LIN {X 0,Y 359.947,Z 582.419,A -85,B 0,C 180,E1 -13482.824,E2 -13482.824} C_VEL
LIN {X 0,Y 358.594,Z 592.161,A -85,B 0,C 180,E1 -13484.075,E2 -13484.075} C_VEL
LIN {X 0,Y 357.358,Z 601.086,A -85,B 0,C 180,E1 -13485.478,E2 -13485.478} C_VEL
LIN {X 0,Y 356.154,Z 609.872,A -85,B 0,C 180,E1 -13487.174,E2 -13487.174} C_VEL
LIN {X 0,Y 355.202,Z 616.932,A -85,B 0,C 180,E1 -13488.877,E2 -13488.877} C_VEL
LIN {X 0,Y 354.322,Z 623.413,A -85,B 0,C 180,E1 -13490.87,E2 -13490.87} C_VEL
LIN {X 0,Y 353.781,Z 627.649,A -85,B 0,C 180,E1 -13492.581,E2 -13492.581} C_VEL
LIN {X 0,Y 353.502,Z 630.768,A -85,B 0,C 180,E1 -13494.295,E2 -13494.295} C_VEL
LIN {X 0,Y 353.381,Z 632.27,A -85,B 0,C 180,E1 -13495.437,E2 -13495.437} C_VEL
LIN {X 0,Y 353.229,Z 633.321,A -85,B 0,C 180,E1 -13496.578,E2 -13496.578} C_VEL
LIN {X 0,Y 353.155,Z 633.956,A -85,B 0,C 180,E1 -13497.719,E2 -13497.719} C_VEL
LIN {X 0,Y 353.153,Z 634.14,A -85,B 0,C 180,E1 -13498.86,E2 -13498.86} C_VEL
LIN {X 0,Y 353.146,Z 633.86,A -85,B 0,C 180,E1 -13500,E2 -13500} C_VEL
LIN {X 0,Y 353.151,Z 633.161,A -85,B 0,C 180,E1 -13501.14,E2 -13501.14} C_VEL
LIN {X 0,Y 353.141,Z 632.017,A -85,B 0,C 180,E1 -13502.281,E2 -13502.281} C_VEL
LIN {X 0,Y 353.281,Z 629.42,A -85,B 0,C 180,E1 -13503.993,E2 -13503.993} C_VEL
LIN {X 0,Y 353.393,Z 624.752,A -85,B 0,C 180,E1 -13506.079,E2 -13506.079} C_VEL
LIN {X 0,Y 353.647,Z 618.898,A -85,B 0,C 180,E1 -13507.996,E2 -13507.996} C_VEL
LIN {X 0,Y 354.026,Z 612.126,A -85,B 0,C 180,E1 -13509.715,E2 -13509.715} C_VEL
LIN {X 0,Y 354.548,Z 603.69,A -85,B 0,C 180,E1 -13511.433,E2 -13511.433} C_VEL
LIN {X 0,Y 355.239,Z 595.006,A -85,B 0,C 180,E1 -13512.86,E2 -13512.86} C_VEL
LIN {X 0,Y 356,Z 584.552,A -85,B 0,C 180,E1 -13514.264,E2 -13514.264} C_VEL
LIN {X 0,Y 356.698,Z 573.904,A -85,B 0,C 180,E1 -13515.425,E2 -13515.425} C_VEL
LIN {X 0,Y 357.436,Z 562.446,A -85,B 0,C 180,E1 -13516.418,E2 -13516.418} C_VEL
LIN {X 0,Y 358.135,Z 549.906,A -85,B 0,C 180,E1 -13517.266,E2 -13517.266} C_VEL
LIN {X 0,Y 358.795,Z 536.113,A -85,B 0,C 180,E1 -13517.933,E2 -13517.933} C_VEL
LIN {X 0,Y 359.155,Z 522.822,A -85,B 0,C 180,E1 -13518.356,E2 -13518.356} C_VEL
LIN {X 0,Y 361.016,Z 446.902,A -85,B 0,C 180,E1 -13520.357,E2 -13520.357} C_VEL
LIN {X 0,Y 357.928,Z 420.522,A -85,B 0,C 180,E1 -13521.225,E2 -13521.225} C_VEL
LIN {X 0,Y 359.275,Z 398.729,A -85,B 0,C 180,E1 -13524.871,E2 -13524.871} C_VEL
LIN {X 0,Y 360.508,Z 380.834,A -85,B 0,C 180,E1 -13527.897,E2 -13527.897} C_VEL
LIN {X 0,Y 358.657,Z 371.766,A -85,B 0,C 180,E1 -13529.579,E2 -13529.579} C_VEL
LIN {X 0,Y 354.853,Z 355.064,A -85,B 0,C 180,E1 -13532.79,E2 -13532.79} C_VEL
LIN {X 0,Y 354.803,Z 354.916,A -85,B 0,C 180,E1 -13536.459,E2 -13536.459} C_VEL
LIN {X 0,Y 354.83,Z 354.91,A -85,B 0,C 180,E1 -13539.423,E2 -13539.423} C_VEL
LIN {X 0,Y 354.794,Z 354.909,A -85,B 0,C 180,E1 -13542.867,E2 -13542.867} C_VEL
LIN {X 0,Y 354.772,Z 354.901,A -85,B 0,C 180,E1 -13546.103,E2 -13546.103} C_VEL
LIN {X 0,Y 354.793,Z 354.906,A -85,B 0,C 180,E1 -13549.178,E2 -13549.178} C_VEL
LIN {X 0,Y 354.818,Z 354.914,A -85,B 0,C 180,E1 -13552.401,E2 -13552.401} C_VEL
LIN {X 0,Y 354.818,Z 354.904,A -85,B 0,C 180,E1 -13554.94,E2 -13554.94} C_VEL
LIN {X 0,Y 354.862,Z 355.109,A -85,B 0,C 180,E1 -13557.978,E2 -13557.978} C_VEL
LIN {X 0,Y 357.702,Z 366.862,A -85,B 0,C 180,E1 -13561.224,E2 -13561.224} C_VEL
LIN {X 0,Y 358.904,Z 372.282,A -85,B 0,C 180,E1 -13562.587,E2 -13562.587} C_VEL
LIN {X 0,Y 364.389,Z 385.82,A -85,B 0,C 180,E1 -13563.36,E2 -13563.36} C_VEL
LIN {X 0,Y 368.616,Z 408.354,A -85,B 0,C 180,E1 -13564.169,E2 -13564.169} C_VEL
LIN {X 0,Y 366.369,Z 509.389,A -85,B 0,C 180,E1 -13566.168,E2 -13566.168} C_VEL
LIN {X 0,Y 365.587,Z 523.29,A -85,B 0,C 180,E1 -13566.64,E2 -13566.64} C_VEL
LIN {X 0,Y 364.552,Z 536.896,A -85,B 0,C 180,E1 -13567.32,E2 -13567.32} C_VEL
LIN {X 0,Y 363.46,Z 549.268,A -85,B 0,C 180,E1 -13568.148,E2 -13568.148} C_VEL
LIN {X 0,Y 362.067,Z 562.159,A -85,B 0,C 180,E1 -13569.251,E2 -13569.251} C_VEL
LIN {X 0,Y 360.6,Z 573.883,A -85,B 0,C 180,E1 -13570.501,E2 -13570.501} C_VEL
LIN {X 0,Y 359.222,Z 583.634,A -85,B 0,C 180,E1 -13571.757,E2 -13571.757} C_VEL
LIN {X 0,Y 357.681,Z 594.412,A -85,B 0,C 180,E1 -13573.445,E2 -13573.445} C_VEL
LIN {X 0,Y 356.413,Z 603.31,A -85,B 0,C 180,E1 -13575.145,E2 -13575.145} C_VEL
LIN {X 0,Y 355.536,Z 610.715,A -85,B 0,C 180,E1 -13576.859,E2 -13576.859} C_VEL
LIN {X 0,Y 354.619,Z 616.889,A -85,B 0,C 180,E1 -13578.568,E2 -13578.568} C_VEL
LIN {X 0,Y 354.047,Z 621.993,A -85,B 0,C 180,E1 -13580.285,E2 -13580.285} C_VEL
LIN {X 0,Y 353.522,Z 627.283,A -85,B 0,C 180,E1 -13582.574,E2 -13582.574} C_VEL
LIN {X 0,Y 353.346,Z 630.234,A -85,B 0,C 180,E1 -13584.291,E2 -13584.291} C_VEL
LIN {X 0,Y 353.206,Z 632.951,A -85,B 0,C 180,E1 -13586.576,E2 -13586.576} C_VEL
LIN {X 0,Y 353.147,Z 634.314,A -85,B 0,C 180,E1 -13588.858,E2 -13588.858} C_VEL
LIN {X 0,Y 353.146,Z 634.35,A -85,B 0,C 180,E1 -13591.139,E2 -13591.139} C_VEL
LIN {X 0,Y 353.204,Z 633.056,A -85,B 0,C 180,E1 -13593.421,E2 -13593.421} C_VEL
LIN {X 0,Y 353.21,Z 632.81,A -85,B 0,C 180,E1 -13593.664,E2 -13593.664} C_VEL
LIN {X 0,Y 352.581,Z 631.862,A -85,B 0,C 180,E1 -13594.603,E2 -13594.603} C_VEL
LIN {X 0,Y 349.808,Z 629.846,A -85,B 0,C 180,E1 -13596.124,E2 -13596.124} C_VEL
LIN {X 0,Y 347.53,Z 627.866,A -85,B 0,C 180,E1 -13597.339,E2 -13597.339} C_VEL
LIN {X 0,Y 346.667,Z 626.094,A -85,B 0,C 180,E1 -13598.265,E2 -13598.265} C_VEL
LIN {X 0,Y 346.659,Z 625.43,A -85,B 0,C 180,E1 -13598.575,E2 -13598.575} C_VEL
LIN {X 0,Y 347.207,Z 620.672,A -85,B 0,C 180,E1 -13600.495,E2 -13600.495} C_VEL
LIN {X 0,Y 348.076,Z 614.308,A -85,B 0,C 180,E1 -13602.534,E2 -13602.534} C_VEL
LIN {X 0,Y 349.119,Z 606.678,A -85,B 0,C 180,E1 -13604.504,E2 -13604.504} C_VEL
LIN {X 0,Y 350.354,Z 598.119,A -85,B 0,C 180,E1 -13606.308,E2 -13606.308} C_VEL
LIN {X 0,Y 351.808,Z 588.15,A -85,B 0,C 180,E1 -13608.036,E2 -13608.036} C_VEL
LIN {X 0,Y 353.433,Z 577.053,A -85,B 0,C 180,E1 -13609.605,E2 -13609.605} C_VEL
LIN {X 0,Y 355.117,Z 564.741,A -85,B 0,C 180,E1 -13611.005,E2 -13611.005} C_VEL
LIN {X 0,Y 356.611,Z 552.281,A -85,B 0,C 180,E1 -13612.14,E2 -13612.14} C_VEL
LIN {X 0,Y 357.796,Z 539.741,A -85,B 0,C 180,E1 -13613.046,E2 -13613.046} C_VEL
LIN {X 0,Y 358.938,Z 526.216,A -85,B 0,C 180,E1 -13613.778,E2 -13613.778} C_VEL
LIN {X 0,Y 359.775,Z 512.644,A -85,B 0,C 180,E1 -13614.294,E2 -13614.294} C_VEL
LIN {X 0,Y 360.395,Z 492.639,A -85,B 0,C 180,E1 -13614.748,E2 -13614.748} C_VEL
LIN {X 0,Y 362.266,Z 408.78,A -85,B 0,C 180,E1 -13616.416,E2 -13616.416} C_VEL
LIN {X 0,Y 358.06,Z 387.656,A -85,B 0,C 180,E1 -13617.216,E2 -13617.216} C_VEL
LIN {X 0,Y 351.708,Z 372.333,A -85,B 0,C 180,E1 -13618.127,E2 -13618.127} C_VEL
LIN {X 0,Y 349.94,Z 364.698,A -85,B 0,C 180,E1 -13620.136,E2 -13620.136} C_VEL
LIN {X 0,Y 347.772,Z 355.882,A -85,B 0,C 180,E1 -13622.694,E2 -13622.694} C_VEL
LIN {X 0,Y 347.767,Z 355.778,A -85,B 0,C 180,E1 -13626.064,E2 -13626.064} C_VEL
LIN {X 0,Y 347.78,Z 355.771,A -85,B 0,C 180,E1 -13629.833,E2 -13629.833} C_VEL
LIN {X 0,Y 347.813,Z 355.777,A -85,B 0,C 180,E1 -13633.392,E2 -13633.392} C_VEL
LIN {X 0,Y 347.811,Z 355.771,A -85,B 0,C 180,E1 -13636.669,E2 -13636.669} C_VEL
LIN {X 0,Y 347.778,Z 355.776,A -85,B 0,C 180,E1 -13640.164,E2 -13640.164} C_VEL
LIN {X 0,Y 347.781,Z 355.77,A -85,B 0,C 180,E1 -13644.124,E2 -13644.124} C_VEL
LIN {X 0,Y 347.73,Z 355.784,A -85,B 0,C 180,E1 -13648.085,E2 -13648.085} C_VEL
LIN {X 0,Y 347.796,Z 355.737,A -85,B 0,C 180,E1 -13650.989,E2 -13650.989} C_VEL
LIN {X 0,Y 347.822,Z 355.765,A -85,B 0,C 180,E1 -13653.607,E2 -13653.607} C_VEL
LIN {X 0,Y 347.779,Z 355.788,A -85,B 0,C 180,E1 -13656.161,E2 -13656.161} C_VEL
LIN {X 0,Y 347.807,Z 355.779,A -85,B 0,C 180,E1 -13659.909,E2 -13659.909} C_VEL
LIN {X 0,Y 347.856,Z 355.775,A -85,B 0,C 180,E1 -13662.359,E2 -13662.359} C_VEL
LIN {X 0,Y 347.887,Z 355.77,A -85,B 0,C 180,E1 -13665.97,E2 -13665.97} C_VEL
LIN {X 0,Y 347.923,Z 355.756,A -85,B 0,C 180,E1 -13669.525,E2 -13669.525} C_VEL
LIN {X 0,Y 348.064,Z 355.747,A -85,B 0,C 180,E1 -13671.874,E2 -13671.874} C_VEL
LIN {X 0,Y 348.058,Z 355.751,A -85,B 0,C 180,E1 -13674.205,E2 -13674.205} C_VEL
LIN {X 0,Y 348.199,Z 355.725,A -85,B 0,C 180,E1 -13677.686,E2 -13677.686} C_VEL
LIN {X 0,Y 348.36,Z 355.715,A -85,B 0,C 180,E1 -13680,E2 -13680} C_VEL
LIN {X 0,Y 348.199,Z 355.726,A -85,B 0,C 180,E1 -13682.313,E2 -13682.313} C_VEL
LIN {X 0,Y 348.096,Z 355.748,A -85,B 0,C 180,E1 -13686.958,E2 -13686.958} C_VEL
LIN {X 0,Y 347.958,Z 355.747,A -85,B 0,C 180,E1 -13689.299,E2 -13689.299} C_VEL
LIN {X 0,Y 347.883,Z 355.774,A -85,B 0,C 180,E1 -13692.84,E2 -13692.84} C_VEL
LIN {X 0,Y 347.828,Z 355.766,A -85,B 0,C 180,E1 -13696.432,E2 -13696.432} C_VEL
LIN {X 0,Y 347.846,Z 355.778,A -85,B 0,C 180,E1 -13698.861,E2 -13698.861} C_VEL
LIN {X 0,Y 347.764,Z 355.783,A -85,B 0,C 180,E1 -13702.58,E2 -13702.58} C_VEL
LIN {X 0,Y 347.802,Z 355.78,A -85,B 0,C 180,E1 -13705.109,E2 -13705.109} C_VEL
LIN {X 0,Y 347.792,Z 355.748,A -85,B 0,C 180,E1 -13707.695,E2 -13707.695} C_VEL
LIN {X 0,Y 347.735,Z 355.756,A -85,B 0,C 180,E1 -13710.349,E2 -13710.349} C_VEL
LIN {X 0,Y 347.739,Z 355.796,A -85,B 0,C 180,E1 -13714.045,E2 -13714.045} C_VEL
LIN {X 0,Y 347.754,Z 355.756,A -85,B 0,C 180,E1 -13717.322,E2 -13717.322} C_VEL
LIN {X 0,Y 347.786,Z 355.779,A -85,B 0,C 180,E1 -13720.29,E2 -13720.29} C_VEL
LIN {X 0,Y 347.812,Z 355.77,A -85,B 0,C 180,E1 -13723.394,E2 -13723.394} C_VEL
LIN {X 0,Y 347.811,Z 355.778,A -85,B 0,C 180,E1 -13726.671,E2 -13726.671} C_VEL
LIN {X 0,Y 347.779,Z 355.771,A -85,B 0,C 180,E1 -13730.167,E2 -13730.167} C_VEL
LIN {X 0,Y 347.784,Z 355.776,A -85,B 0,C 180,E1 -13734.126,E2 -13734.126} C_VEL
LIN {X 0,Y 347.779,Z 355.927,A -85,B 0,C 180,E1 -13737.385,E2 -13737.385} C_VEL
LIN {X 0,Y 350.564,Z 367.135,A -85,B 0,C 180,E1 -13740.585,E2 -13740.585} C_VEL
LIN {X 0,Y 351.713,Z 372.239,A -85,B 0,C 180,E1 -13741.909,E2 -13741.909} C_VEL
LIN {X 0,Y 358.251,Z 388.211,A -85,B 0,C 180,E1 -13742.857,E2 -13742.857} C_VEL
LIN {X 0,Y 362.277,Z 409.098,A -85,B 0,C 180,E1 -13743.637,E2 -13743.637} C_VEL
LIN {X 0,Y 359.967,Z 508.981,A -85,B 0,C 180,E1 -13745.643,E2 -13745.643} C_VEL
LIN {X 0,Y 359.109,Z 523.036,A -85,B 0,C 180,E1 -13746.119,E2 -13746.119} C_VEL
LIN {X 0,Y 358.035,Z 536.704,A -85,B 0,C 180,E1 -13746.81,E2 -13746.81} C_VEL
LIN {X 0,Y 356.775,Z 550.651,A -85,B 0,C 180,E1 -13747.776,E2 -13747.776} C_VEL
LIN {X 0,Y 355.411,Z 562.942,A -85,B 0,C 180,E1 -13748.867,E2 -13748.867} C_VEL
LIN {X 0,Y 353.846,Z 574.376,A -85,B 0,C 180,E1 -13750.117,E2 -13750.117} C_VEL
LIN {X 0,Y 352.148,Z 585.994,A -85,B 0,C 180,E1 -13751.681,E2 -13751.681} C_VEL
LIN {X 0,Y 350.585,Z 596.381,A -85,B 0,C 180,E1 -13753.403,E2 -13753.403} C_VEL
LIN {X 0,Y 349.353,Z 604.834,A -85,B 0,C 180,E1 -13755.114,E2 -13755.114} C_VEL
LIN {X 0,Y 348.25,Z 613.149,A -85,B 0,C 180,E1 -13757.176,E2 -13757.176} C_VEL
LIN {X 0,Y 347.393,Z 618.887,A -85,B 0,C 180,E1 -13758.921,E2 -13758.921} C_VEL
LIN {X 0,Y 346.852,Z 623.587,A -85,B 0,C 180,E1 -13760.673,E2 -13760.673} C_VEL
LIN {X 0,Y 346.412,Z 628.461,A -85,B 0,C 180,E1 -13763.01,E2 -13763.01} C_VEL
LIN {X 0,Y 346.211,Z 631.845,A -85,B 0,C 180,E1 -13765.344,E2 -13765.344} C_VEL
LIN {X 0,Y 346.049,Z 633.842,A -85,B 0,C 180,E1 -13767.674,E2 -13767.674} C_VEL
LIN {X 0,Y 346.044,Z 634.5,A -85,B 0,C 180,E1 -13770.001,E2 -13770.001} C_VEL
LIN {X 0,Y 346.049,Z 633.83,A -85,B 0,C 180,E1 -13772.329,E2 -13772.329} C_VEL
LIN {X 0,Y 346.204,Z 631.821,A -85,B 0,C 180,E1 -13774.659,E2 -13774.659} C_VEL
LIN {X 0,Y 346.375,Z 628.429,A -85,B 0,C 180,E1 -13776.994,E2 -13776.994} C_VEL
LIN {X 0,Y 346.855,Z 623.549,A -85,B 0,C 180,E1 -13779.33,E2 -13779.33} C_VEL
LIN {X 0,Y 347.395,Z 618.838,A -85,B 0,C 180,E1 -13781.082,E2 -13781.082} C_VEL
LIN {X 0,Y 348.406,Z 612.002,A -85,B 0,C 180,E1 -13783.118,E2 -13783.118} C_VEL
LIN {X 0,Y 349.499,Z 603.517,A -85,B 0,C 180,E1 -13785.155,E2 -13785.155} C_VEL
LIN {X 0,Y 350.816,Z 594.659,A -85,B 0,C 180,E1 -13786.888,E2 -13786.888} C_VEL
LIN {X 0,Y 352.415,Z 583.928,A -85,B 0,C 180,E1 -13788.609,E2 -13788.609} C_VEL
LIN {X 0,Y 354.006,Z 573.063,A -85,B 0,C 180,E1 -13790.028,E2 -13790.028} C_VEL
LIN {X 0,Y 355.686,Z 560.281,A -85,B 0,C 180,E1 -13791.384,E2 -13791.384} C_VEL
LIN {X 0,Y 356.945,Z 548.533,A -85,B 0,C 180,E1 -13792.381,E2 -13792.381} C_VEL
LIN {X 0,Y 358.136,Z 535.285,A -85,B 0,C 180,E1 -13793.263,E2 -13793.263} C_VEL
LIN {X 0,Y 359.222,Z 520.896,A -85,B 0,C 180,E1 -13793.953,E2 -13793.953} C_VEL
LIN {X 0,Y 359.942,Z 506.766,A -85,B 0,C 180,E1 -13794.4,E2 -13794.4} C_VEL
LIN {X 0,Y 362.245,Z 409.751,A -85,B 0,C 180,E1 -13796.335,E2 -13796.335} C_VEL
LIN {X 0,Y 361.769,Z 405.943,A -85,B 0,C 180,E1 -13796.478,E2 -13796.478} C_VEL
LIN {X 0,Y 362.438,Z 393.312,A -85,B 0,C 180,E1 -13797.736,E2 -13797.736} C_VEL
LIN {X 0,Y 361.547,Z 388.45,A -85,B 0,C 180,E1 -13798.512,E2 -13798.512} C_VEL
LIN {X 0,Y 358.725,Z 376.947,A -85,B 0,C 180,E1 -13800.867,E2 -13800.867} C_VEL
LIN {X 0,Y 357.981,Z 374.036,A -85,B 0,C 180,E1 -13801.596,E2 -13801.596} C_VEL
LIN {X 0,Y 356.171,Z 370.514,A -85,B 0,C 180,E1 -13802.865,E2 -13802.865} C_VEL
LIN {X 0,Y 353.211,Z 365.674,A -85,B 0,C 180,E1 -13805.334,E2 -13805.334} C_VEL
LIN {X 0,Y 351.771,Z 363.551,A -85,B 0,C 180,E1 -13806.95,E2 -13806.95} C_VEL
LIN {X 0,Y 350.883,Z 361.791,A -85,B 0,C 180,E1 -13808.634,E2 -13808.634} C_VEL
LIN {X 0,Y 350.452,Z 360.661,A -85,B 0,C 180,E1 -13810.354,E2 -13810.354} C_VEL
LIN {X 0,Y 350.366,Z 360.594,A -85,B 0,C 180,E1 -13813.002,E2 -13813.002} C_VEL
LIN {X 0,Y 350.819,Z 362.288,A -85,B 0,C 180,E1 -13815.48,E2 -13815.48} C_VEL
LIN {X 0,Y 352.401,Z 364.88,A -85,B 0,C 180,E1 -13818.036,E2 -13818.036} C_VEL
LIN {X 0,Y 354.302,Z 369.465,A -85,B 0,C 180,E1 -13820.681,E2 -13820.681} C_VEL
LIN {X 0,Y 356.403,Z 374.91,A -85,B 0,C 180,E1 -13823.081,E2 -13823.081} C_VEL
LIN {X 0,Y 358.542,Z 381.47,A -85,B 0,C 180,E1 -13825.415,E2 -13825.415} C_VEL
LIN {X 0,Y 360.488,Z 389.176,A -85,B 0,C 180,E1 -13827.695,E2 -13827.695} C_VEL
LIN {X 0,Y 361.638,Z 395.793,A -85,B 0,C 180,E1 -13829.402,E2 -13829.402} C_VEL
LIN {X 0,Y 361.647,Z 398.432,A -85,B 0,C 180,E1 -13829.973,E2 -13829.973} C_VEL
LIN {X 0,Y 358.615,Z 419.509,A -85,B 0,C 180,E1 -13833.859,E2 -13833.859} C_VEL
LIN {X 0,Y 360.523,Z 429.198,A -85,B 0,C 180,E1 -13834.641,E2 -13834.641} C_VEL
LIN {X 0,Y 363.201,Z 444.906,A -85,B 0,C 180,E1 -13835.674,E2 -13835.674} C_VEL
LIN {X 0,Y 363.881,Z 452.419,A -85,B 0,C 180,E1 -13836.072,E2 -13836.072} C_VEL
LIN {X 0,Y 358.846,Z 534.111,A -85,B 0,C 180,E1 -13838.682,E2 -13838.682} C_VEL
LIN {X 0,Y 357.61,Z 548.003,A -85,B 0,C 180,E1 -13839.358,E2 -13839.358} C_VEL
LIN {X 0,Y 356.434,Z 559.425,A -85,B 0,C 180,E1 -13840.115,E2 -13840.115} C_VEL
LIN {X 0,Y 355.043,Z 570.896,A -85,B 0,C 180,E1 -13841.087,E2 -13841.087} C_VEL
LIN {X 0,Y 353.481,Z 582.749,A -85,B 0,C 180,E1 -13842.35,E2 -13842.35} C_VEL
LIN {X 0,Y 351.868,Z 593.345,A -85,B 0,C 180,E1 -13843.762,E2 -13843.762} C_VEL
LIN {X 0,Y 350.555,Z 602.063,A -85,B 0,C 180,E1 -13845.19,E2 -13845.19} C_VEL
LIN {X 0,Y 349.427,Z 609.329,A -85,B 0,C 180,E1 -13846.627,E2 -13846.627} C_VEL
LIN {X 0,Y 348.482,Z 616.497,A -85,B 0,C 180,E1 -13848.365,E2 -13848.365} C_VEL
LIN {X 0,Y 347.569,Z 622.23,A -85,B 0,C 180,E1 -13850.103,E2 -13850.103} C_VEL
LIN {X 0,Y 346.879,Z 626.729,A -85,B 0,C 180,E1 -13851.847,E2 -13851.847} C_VEL
LIN {X 0,Y 346.508,Z 630.172,A -85,B 0,C 180,E1 -13853.643,E2 -13853.643} C_VEL
LIN {X 0,Y 346.301,Z 632.427,A -85,B 0,C 180,E1 -13855.344,E2 -13855.344} C_VEL
LIN {X 0,Y 346.158,Z 633.428,A -85,B 0,C 180,E1 -13856.508,E2 -13856.508} C_VEL
LIN {X 0,Y 346.069,Z 634.005,A -85,B 0,C 180,E1 -13857.672,E2 -13857.672} C_VEL
LIN {X 0,Y 346.056,Z 634.1,A -85,B 0,C 180,E1 -13858.836,E2 -13858.836} C_VEL
LIN {X 0,Y 346.048,Z 633.771,A -85,B 0,C 180,E1 -13860,E2 -13860} C_VEL
LIN {X 0,Y 346.054,Z 633.019,A -85,B 0,C 180,E1 -13861.164,E2 -13861.164} C_VEL
LIN {X 0,Y 346.055,Z 631.778,A -85,B 0,C 180,E1 -13862.328,E2 -13862.328} C_VEL
LIN {X 0,Y 346.215,Z 629.077,A -85,B 0,C 180,E1 -13864.074,E2 -13864.074} C_VEL
LIN {X 0,Y 346.292,Z 624.738,A -85,B 0,C 180,E1 -13866.028,E2 -13866.028} C_VEL
LIN {X 0,Y 346.488,Z 620.216,A -85,B 0,C 180,E1 -13867.576,E2 -13867.576} C_VEL
LIN {X 0,Y 346.815,Z 613.818,A -85,B 0,C 180,E1 -13869.33,E2 -13869.33} C_VEL
LIN {X 0,Y 347.324,Z 605.754,A -85,B 0,C 180,E1 -13871.083,E2 -13871.083} C_VEL
LIN {X 0,Y 347.974,Z 597.525,A -85,B 0,C 180,E1 -13872.54,E2 -13872.54} C_VEL
LIN {X 0,Y 348.669,Z 588.61,A -85,B 0,C 180,E1 -13873.849,E2 -13873.849} C_VEL
LIN {X 0,Y 349.42,Z 577.706,A -85,B 0,C 180,E1 -13875.158,E2 -13875.158} C_VEL
LIN {X 0,Y 350.159,Z 565.545,A -85,B 0,C 180,E1 -13876.32,E2 -13876.32} C_VEL
LIN {X 0,Y 350.927,Z 552.784,A -85,B 0,C 180,E1 -13877.257,E2 -13877.257} C_VEL
LIN {X 0,Y 351.643,Z 538.834,A -85,B 0,C 180,E1 -13878.009,E2 -13878.009} C_VEL
LIN {X 0,Y 352.12,Z 525.828,A -85,B 0,C 180,E1 -13878.473,E2 -13878.473} C_VEL
LIN {X 0,Y 354.138,Z 447.749,A -85,B 0,C 180,E1 -13880.59,E2 -13880.59} C_VEL
LIN {X 0,Y 351.036,Z 421.382,A -85,B 0,C 180,E1 -13881.47,E2 -13881.47} C_VEL
LIN {X 0,Y 351.008,Z 419.931,A -85,B 0,C 180,E1 -13881.587,E2 -13881.587} C_VEL
LIN {X 0,Y 352.355,Z 399.455,A -85,B 0,C 180,E1 -13885.078,E2 -13885.078} C_VEL
LIN {X 0,Y 353.535,Z 383.276,A -85,B 0,C 180,E1 -13887.85,E2 -13887.85} C_VEL
LIN {X 0,Y 353.178,Z 379.518,A -85,B 0,C 180,E1 -13888.528,E2 -13888.528} C_VEL
LIN {X 0,Y 348.801,Z 360.326,A -85,B 0,C 180,E1 -13892.191,E2 -13892.191} C_VEL
LIN {X 0,Y 347.796,Z 355.914,A -85,B 0,C 180,E1 -13893.106,E2 -13893.106} C_VEL
LIN {X 0,Y 347.776,Z 355.791,A -85,B 0,C 180,E1 -13896.065,E2 -13896.065} C_VEL
LIN {X 0,Y 347.758,Z 355.792,A -85,B 0,C 180,E1 -13898.792,E2 -13898.792} C_VEL
LIN {X 0,Y 347.756,Z 355.793,A -85,B 0,C 180,E1 -13901.83,E2 -13901.83} C_VEL
LIN {X 0,Y 347.71,Z 355.771,A -85,B 0,C 180,E1 -13905.026,E2 -13905.026} C_VEL
LIN {X 0,Y 347.756,Z 355.79,A -85,B 0,C 180,E1 -13908.396,E2 -13908.396} C_VEL
LIN {X 0,Y 347.783,Z 355.788,A -85,B 0,C 180,E1 -13912.01,E2 -13912.01} C_VEL
LIN {X 0,Y 347.75,Z 355.792,A -85,B 0,C 180,E1 -13915.535,E2 -13915.535} C_VEL
LIN {X 0,Y 347.78,Z 355.848,A -85,B 0,C 180,E1 -13917.389,E2 -13917.389} C_VEL
LIN {X 0,Y 349.183,Z 361.638,A -85,B 0,C 180,E1 -13919.12,E2 -13919.12} C_VEL
LIN {X 0,Y 351.584,Z 371.806,A -85,B 0,C 180,E1 -13921.888,E2 -13921.888} C_VEL
LIN {X 0,Y 351.927,Z 373.035,A -85,B 0,C 180,E1 -13922.038,E2 -13922.038} C_VEL
LIN {X 0,Y 358.298,Z 388.418,A -85,B 0,C 180,E1 -13922.928,E2 -13922.928} C_VEL
LIN {X 0,Y 362.237,Z 409.252,A -85,B 0,C 180,E1 -13923.698,E2 -13923.698} C_VEL
LIN {X 0,Y 359.911,Z 509.406,A -85,B 0,C 180,E1 -13925.713,E2 -13925.713} C_VEL
LIN {X 0,Y 359.086,Z 523.301,A -85,B 0,C 180,E1 -13926.191,E2 -13926.191} C_VEL
LIN {X 0,Y 358.015,Z 536.904,A -85,B 0,C 180,E1 -13926.882,E2 -13926.882} C_VEL
LIN {X 0,Y 356.75,Z 550.316,A -85,B 0,C 180,E1 -13927.805,E2 -13927.805} C_VEL
LIN {X 0,Y 355.236,Z 563.633,A -85,B 0,C 180,E1 -13928.99,E2 -13928.99} C_VEL
LIN {X 0,Y 353.698,Z 575.061,A -85,B 0,C 180,E1 -13930.256,E2 -13930.256} C_VEL
LIN {X 0,Y 352.18,Z 585.587,A -85,B 0,C 180,E1 -13931.68,E2 -13931.68} C_VEL
LIN {X 0,Y 350.613,Z 596.042,A -85,B 0,C 180,E1 -13933.402,E2 -13933.402} C_VEL
LIN {X 0,Y 349.36,Z 604.549,A -85,B 0,C 180,E1 -13935.111,E2 -13935.111} C_VEL
LIN {X 0,Y 348.26,Z 612.934,A -85,B 0,C 180,E1 -13937.173,E2 -13937.173} C_VEL
LIN {X 0,Y 347.435,Z 618.7,A -85,B 0,C 180,E1 -13938.919,E2 -13938.919} C_VEL
LIN {X 0,Y 346.862,Z 623.44,A -85,B 0,C 180,E1 -13940.67,E2 -13940.67} C_VEL
LIN {X 0,Y 346.377,Z 628.347,A -85,B 0,C 180,E1 -13943.006,E2 -13943.006} C_VEL
LIN {X 0,Y 346.209,Z 631.765,A -85,B 0,C 180,E1 -13945.341,E2 -13945.341} C_VEL
LIN {X 0,Y 346.051,Z 633.799,A -85,B 0,C 180,E1 -13947.671,E2 -13947.671} C_VEL
LIN {X 0,Y 346.045,Z 634.498,A -85,B 0,C 180,E1 -13949.999,E2 -13949.999} C_VEL
LIN {X 0,Y 346.05,Z 633.87,A -85,B 0,C 180,E1 -13952.326,E2 -13952.326} C_VEL
LIN {X 0,Y 346.203,Z 631.901,A -85,B 0,C 180,E1 -13954.656,E2 -13954.656} C_VEL
LIN {X 0,Y 346.411,Z 628.543,A -85,B 0,C 180,E1 -13956.99,E2 -13956.99} C_VEL
LIN {X 0,Y 346.659,Z 625.43,A -85,B 0,C 180,E1 -13958.575,E2 -13958.575} C_VEL
LIN {X 0,Y 346.238,Z 623.403,A -85,B 0,C 180,E1 -13959.489,E2 -13959.489} C_VEL
LIN {X 0,Y 343.844,Z 619.742,A -85,B 0,C 180,E1 -13960.967,E2 -13960.967} C_VEL
LIN {X 0,Y 341.588,Z 615.517,A -85,B 0,C 180,E1 -13962.421,E2 -13962.421} C_VEL
LIN {X 0,Y 341.388,Z 612.606,A -85,B 0,C 180,E1 -13963.284,E2 -13963.284} C_VEL
LIN {X 0,Y 342.549,Z 604.286,A -85,B 0,C 180,E1 -13965.357,E2 -13965.357} C_VEL
LIN {X 0,Y 343.98,Z 594.996,A -85,B 0,C 180,E1 -13967.231,E2 -13967.231} C_VEL
LIN {X 0,Y 345.624,Z 584.331,A -85,B 0,C 180,E1 -13968.985,E2 -13968.985} C_VEL
LIN {X 0,Y 347.275,Z 573.547,A -85,B 0,C 180,E1 -13970.43,E2 -13970.43} C_VEL
LIN {X 0,Y 348.781,Z 562.448,A -85,B 0,C 180,E1 -13971.654,E2 -13971.654} C_VEL
LIN {X 0,Y 350.339,Z 549.417,A -85,B 0,C 180,E1 -13972.809,E2 -13972.809} C_VEL
LIN {X 0,Y 351.584,Z 536.231,A -85,B 0,C 180,E1 -13973.72,E2 -13973.72} C_VEL
LIN {X 0,Y 352.727,Z 522.371,A -85,B 0,C 180,E1 -13974.419,E2 -13974.419} C_VEL
LIN {X 0,Y 353.487,Z 509.187,A -85,B 0,C 180,E1 -13974.872,E2 -13974.872} C_VEL
LIN {X 0,Y 355.941,Z 409.996,A -85,B 0,C 180,E1 -13976.896,E2 -13976.896} C_VEL
LIN {X 0,Y 352.012,Z 390.296,A -85,B 0,C 180,E1 -13977.664,E2 -13977.664} C_VEL
LIN {X 0,Y 344.527,Z 372.43,A -85,B 0,C 180,E1 -13978.76,E2 -13978.76} C_VEL
LIN {X 0,Y 343.658,Z 368.74,A -85,B 0,C 180,E1 -13979.698,E2 -13979.698} C_VEL
LIN {X 0,Y 341.091,Z 358.287,A -85,B 0,C 180,E1 -13982.705,E2 -13982.705} C_VEL
LIN {X 0,Y 340.72,Z 356.686,A -85,B 0,C 180,E1 -13983.287,E2 -13983.287} C_VEL
LIN {X 0,Y 340.703,Z 356.662,A -85,B 0,C 180,E1 -13986.74,E2 -13986.74} C_VEL
LIN {X 0,Y 340.759,Z 356.646,A -85,B 0,C 180,E1 -13990.261,E2 -13990.261} C_VEL
LIN {X 0,Y 340.773,Z 356.647,A -85,B 0,C 180,E1 -13993.794,E2 -13993.794} C_VEL
LIN {X 0,Y 340.754,Z 356.656,A -85,B 0,C 180,E1 -13997.108,E2 -13997.108} C_VEL
LIN {X 0,Y 340.727,Z 356.653,A -85,B 0,C 180,E1 -14000.251,E2 -14000.251} C_VEL
LIN {X 0,Y 340.703,Z 356.643,A -85,B 0,C 180,E1 -14003.558,E2 -14003.558} C_VEL
LIN {X 0,Y 340.686,Z 356.674,A -85,B 0,C 180,E1 -14006.152,E2 -14006.152} C_VEL
LIN {X 0,Y 340.766,Z 356.614,A -85,B 0,C 180,E1 -14010.331,E2 -14010.331} C_VEL
LIN {X 0,Y 340.796,Z 356.633,A -85,B 0,C 180,E1 -14013.019,E2 -14013.019} C_VEL
LIN {X 0,Y 340.719,Z 356.668,A -85,B 0,C 180,E1 -14016.926,E2 -14016.926} C_VEL
LIN {X 0,Y 340.785,Z 356.656,A -85,B 0,C 180,E1 -14020.733,E2 -14020.733} C_VEL
LIN {X 0,Y 340.776,Z 356.651,A -85,B 0,C 180,E1 -14023.218,E2 -14023.218} C_VEL
LIN {X 0,Y 340.837,Z 356.649,A -85,B 0,C 180,E1 -14026.89,E2 -14026.89} C_VEL
LIN {X 0,Y 340.919,Z 356.623,A -85,B 0,C 180,E1 -14030.507,E2 -14030.507} C_VEL
LIN {X 0,Y 341.065,Z 356.621,A -85,B 0,C 180,E1 -14032.898,E2 -14032.898} C_VEL
LIN {X 0,Y 341.16,Z 356.601,A -85,B 0,C 180,E1 -14037.639,E2 -14037.639} C_VEL
LIN {X 0,Y 341.33,Z 356.591,A -85,B 0,C 180,E1 -14040,E2 -14040} C_VEL
LIN {X 0,Y 341.16,Z 356.601,A -85,B 0,C 180,E1 -14042.361,E2 -14042.361} C_VEL
LIN {X 0,Y 341.065,Z 356.622,A -85,B 0,C 180,E1 -14047.102,E2 -14047.102} C_VEL
LIN {X 0,Y 340.865,Z 356.635,A -85,B 0,C 180,E1 -14050.694,E2 -14050.694} C_VEL
LIN {X 0,Y 340.852,Z 356.641,A -85,B 0,C 180,E1 -14054.325,E2 -14054.325} C_VEL
LIN {X 0,Y 340.827,Z 356.653,A -85,B 0,C 180,E1 -14058.467,E2 -14058.467} C_VEL
LIN {X 0,Y 340.743,Z 356.651,A -85,B 0,C 180,E1 -14061.858,E2 -14061.858} C_VEL
LIN {X 0,Y 340.762,Z 356.656,A -85,B 0,C 180,E1 -14065.665,E2 -14065.665} C_VEL
LIN {X 0,Y 340.709,Z 356.62,A -85,B 0,C 180,E1 -14068.322,E2 -14068.322} C_VEL
LIN {X 0,Y 340.686,Z 356.644,A -85,B 0,C 180,E1 -14071.046,E2 -14071.046} C_VEL
LIN {X 0,Y 340.709,Z 356.663,A -85,B 0,C 180,E1 -14075.28,E2 -14075.28} C_VEL
LIN {X 0,Y 340.709,Z 356.633,A -85,B 0,C 180,E1 -14078.389,E2 -14078.389} C_VEL
LIN {X 0,Y 340.72,Z 356.668,A -85,B 0,C 180,E1 -14081.305,E2 -14081.305} C_VEL
LIN {X 0,Y 340.774,Z 356.634,A -85,B 0,C 180,E1 -14084.524,E2 -14084.524} C_VEL
LIN {X 0,Y 340.747,Z 356.667,A -85,B 0,C 180,E1 -14087.946,E2 -14087.946} C_VEL
LIN {X 0,Y 340.728,Z 356.649,A -85,B 0,C 180,E1 -14090.254,E2 -14090.254} C_VEL
LIN {X 0,Y 340.706,Z 356.659,A -85,B 0,C 180,E1 -14093.56,E2 -14093.56} C_VEL
LIN {X 0,Y 340.753,Z 356.824,A -85,B 0,C 180,E1 -14096.872,E2 -14096.872} C_VEL
LIN {X 0,Y 343.632,Z 368.577,A -85,B 0,C 180,E1 -14100.303,E2 -14100.303} C_VEL
LIN {X 0,Y 344.483,Z 372.233,A -85,B 0,C 180,E1 -14101.264,E2 -14101.264} C_VEL
LIN {X 0,Y 351.68,Z 389.266,A -85,B 0,C 180,E1 -14102.33,E2 -14102.33} C_VEL
LIN {X 0,Y 353.309,Z 396.247,A -85,B 0,C 180,E1 -14102.625,E2 -14102.625} C_VEL
LIN {X 0,Y 355.888,Z 409.749,A -85,B 0,C 180,E1 -14103.14,E2 -14103.14} C_VEL
LIN {X 0,Y 353.928,Z 492.355,A -85,B 0,C 180,E1 -14104.808,E2 -14104.808} C_VEL
LIN {X 0,Y 353.306,Z 512.46,A -85,B 0,C 180,E1 -14105.271,E2 -14105.271} C_VEL
LIN {X 0,Y 352.35,Z 526.853,A -85,B 0,C 180,E1 -14105.827,E2 -14105.827} C_VEL
LIN {X 0,Y 351.223,Z 540.325,A -85,B 0,C 180,E1 -14106.583,E2 -14106.583} C_VEL
LIN {X 0,Y 349.858,Z 553.518,A -85,B 0,C 180,E1 -14107.564,E2 -14107.564} C_VEL
LIN {X 0,Y 348.425,Z 565.612,A -85,B 0,C 180,E1 -14108.713,E2 -14108.713} C_VEL
LIN {X 0,Y 346.641,Z 577.811,A -85,B 0,C 180,E1 -14110.149,E2 -14110.149} C_VEL
LIN {X 0,Y 345.093,Z 587.886,A -85,B 0,C 180,E1 -14111.601,E2 -14111.601} C_VEL
LIN {X 0,Y 343.498,Z 597.898,A -85,B 0,C 180,E1 -14113.357,E2 -14113.357} C_VEL
LIN {X 0,Y 342.132,Z 607.024,A -85,B 0,C 180,E1 -14115.324,E2 -14115.324} C_VEL
LIN {X 0,Y 341.147,Z 614.157,A -85,B 0,C 180,E1 -14117.207,E2 -14117.207} C_VEL
LIN {X 0,Y 340.19,Z 620.55,A -85,B 0,C 180,E1 -14119.286,E2 -14119.286} C_VEL
LIN {X 0,Y 339.522,Z 626.219,A -85,B 0,C 180,E1 -14121.67,E2 -14121.67} C_VEL
LIN {X 0,Y 339.208,Z 630.333,A -85,B 0,C 180,E1 -14124.055,E2 -14124.055} C_VEL
LIN {X 0,Y 339.06,Z 633.013,A -85,B 0,C 180,E1 -14126.436,E2 -14126.436} C_VEL
LIN {X 0,Y 338.954,Z 634.337,A -85,B 0,C 180,E1 -14128.813,E2 -14128.813} C_VEL
LIN {X 0,Y 338.954,Z 634.331,A -85,B 0,C 180,E1 -14131.19,E2 -14131.19} C_VEL
LIN {X 0,Y 339.059,Z 632.994,A -85,B 0,C 180,E1 -14133.567,E2 -14133.567} C_VEL
LIN {X 0,Y 339.207,Z 630.214,A -85,B 0,C 180,E1 -14136.008,E2 -14136.008} C_VEL
LIN {X 0,Y 339.525,Z 626.195,A -85,B 0,C 180,E1 -14138.333,E2 -14138.333} C_VEL
LIN {X 0,Y 340.192,Z 620.504,A -85,B 0,C 180,E1 -14140.717,E2 -14140.717} C_VEL
LIN {X 0,Y 341.142,Z 614.096,A -85,B 0,C 180,E1 -14142.796,E2 -14142.796} C_VEL
LIN {X 0,Y 342.138,Z 606.949,A -85,B 0,C 180,E1 -14144.679,E2 -14144.679} C_VEL
LIN {X 0,Y 343.499,Z 597.807,A -85,B 0,C 180,E1 -14146.646,E2 -14146.646} C_VEL
LIN {X 0,Y 345.07,Z 587.775,A -85,B 0,C 180,E1 -14148.404,E2 -14148.404} C_VEL
LIN {X 0,Y 346.802,Z 576.579,A -85,B 0,C 180,E1 -14149.999,E2 -14149.999} C_VEL
LIN {X 0,Y 348.526,Z 564.246,A -85,B 0,C 180,E1 -14151.413,E2 -14151.413} C_VEL
LIN {X 0,Y 349.992,Z 551.706,A -85,B 0,C 180,E1 -14152.57,E2 -14152.57} C_VEL
LIN {X 0,Y 351.336,Z 538.693,A -85,B 0,C 180,E1 -14153.506,E2 -14153.506} C_VEL
LIN {X 0,Y 352.451,Z 525.712,A -85,B 0,C 180,E1 -14154.208,E2 -14154.208} C_VEL
LIN {X 0,Y 353.299,Z 511.877,A -85,B 0,C 180,E1 -14154.733,E2 -14154.733} C_VEL
LIN {X 0,Y 353.998,Z 489.639,A -85,B 0,C 180,E1 -14155.229,E2 -14155.229} C_VEL
LIN {X 0,Y 355.901,Z 411.844,A -85,B 0,C 180,E1 -14156.824,E2 -14156.824} C_VEL
LIN {X 0,Y 356.38,Z 408.076,A -85,B 0,C 180,E1 -14157.125,E2 -14157.125} C_VEL
LIN {X 0,Y 357.25,Z 396.717,A -85,B 0,C 180,E1 -14158.308,E2 -14158.308} C_VEL
LIN {X 0,Y 356.644,Z 392.84,A -85,B 0,C 180,E1 -14158.941,E2 -14158.941} C_VEL
LIN {X 0,Y 354.296,Z 382.683,A -85,B 0,C 180,E1 -14161.049,E2 -14161.049} C_VEL
LIN {X 0,Y 353.479,Z 379.186,A -85,B 0,C 180,E1 -14161.919,E2 -14161.919} C_VEL
LIN {X 0,Y 351.996,Z 376.205,A -85,B 0,C 180,E1 -14163.01,E2 -14163.01} C_VEL
LIN {X 0,Y 349.454,Z 371.997,A -85,B 0,C 180,E1 -14165.108,E2 -14165.108} C_VEL
LIN {X 0,Y 347.165,Z 368.401,A -85,B 0,C 180,E1 -14167.86,E2 -14167.86} C_VEL
LIN {X 0,Y 346.512,Z 366.842,A -85,B 0,C 180,E1 -14169.581,E2 -14169.581} C_VEL
LIN {X 0,Y 346.11,Z 366.225,A -85,B 0,C 180,E1 -14171.296,E2 -14171.296} C_VEL
LIN {X 0,Y 346.154,Z 366.527,A -85,B 0,C 180,E1 -14173.656,E2 -14173.656} C_VEL
LIN {X 0,Y 347.005,Z 369.05,A -85,B 0,C 180,E1 -14176.814,E2 -14176.814} C_VEL
LIN {X 0,Y 347.916,Z 370.906,A -85,B 0,C 180,E1 -14178.368,E2 -14178.368} C_VEL
LIN {X 0,Y 349.492,Z 374.811,A -85,B 0,C 180,E1 -14180.696,E2 -14180.696} C_VEL
LIN {X 0,Y 351.421,Z 380.198,A -85,B 0,C 180,E1 -14183.133,E2 -14183.133} C_VEL
LIN {X 0,Y 353.355,Z 386.643,A -85,B 0,C 180,E1 -14185.464,E2 -14185.464} C_VEL
LIN {X 0,Y 355.218,Z 395.068,A -85,B 0,C 180,E1 -14187.98,E2 -14187.98} C_VEL
LIN {X 0,Y 355.838,Z 400.854,A -85,B 0,C 180,E1 -14189.431,E2 -14189.431} C_VEL
LIN {X 0,Y 352.953,Z 420.055,A -85,B 0,C 180,E1 -14193.032,E2 -14193.032} C_VEL
LIN {X 0,Y 356.026,Z 435.617,A -85,B 0,C 180,E1 -14194.277,E2 -14194.277} C_VEL
LIN {X 0,Y 358.047,Z 449.915,A -85,B 0,C 180,E1 -14195.206,E2 -14195.206} C_VEL
LIN {X 0,Y 358.224,Z 454.652,A -85,B 0,C 180,E1 -14195.437,E2 -14195.437} C_VEL
LIN {X 0,Y 352.848,Z 534.393,A -85,B 0,C 180,E1 -14198.071,E2 -14198.071} C_VEL
LIN {X 0,Y 351.56,Z 548.059,A -85,B 0,C 180,E1 -14198.756,E2 -14198.756} C_VEL
LIN {X 0,Y 350.191,Z 560.277,A -85,B 0,C 180,E1 -14199.592,E2 -14199.592} C_VEL
LIN {X 0,Y 348.705,Z 571.523,A -85,B 0,C 180,E1 -14200.576,E2 -14200.576} C_VEL
LIN {X 0,Y 347.044,Z 583.208,A -85,B 0,C 180,E1 -14201.859,E2 -14201.859} C_VEL
LIN {X 0,Y 345.165,Z 594.635,A -85,B 0,C 180,E1 -14203.438,E2 -14203.438} C_VEL
LIN {X 0,Y 343.798,Z 603.121,A -85,B 0,C 180,E1 -14204.892,E2 -14204.892} C_VEL
LIN {X 0,Y 342.587,Z 610.201,A -85,B 0,C 180,E1 -14206.354,E2 -14206.354} C_VEL
LIN {X 0,Y 341.573,Z 617.145,A -85,B 0,C 180,E1 -14208.126,E2 -14208.126} C_VEL
LIN {X 0,Y 340.595,Z 622.747,A -85,B 0,C 180,E1 -14209.899,E2 -14209.899} C_VEL
LIN {X 0,Y 339.851,Z 627.121,A -85,B 0,C 180,E1 -14211.677,E2 -14211.677} C_VEL
LIN {X 0,Y 339.42,Z 630.699,A -85,B 0,C 180,E1 -14213.668,E2 -14213.668} C_VEL
LIN {X 0,Y 339.225,Z 632.596,A -85,B 0,C 180,E1 -14215.246,E2 -14215.246} C_VEL
LIN {X 0,Y 339.089,Z 633.544,A -85,B 0,C 180,E1 -14216.435,E2 -14216.435} C_VEL
LIN {X 0,Y 338.985,Z 634.022,A -85,B 0,C 180,E1 -14217.624,E2 -14217.624} C_VEL
LIN {X 0,Y 338.962,Z 634.059,A -85,B 0,C 180,E1 -14218.812,E2 -14218.812} C_VEL
LIN {X 0,Y 338.953,Z 633.676,A -85,B 0,C 180,E1 -14220,E2 -14220} C_VEL
LIN {X 0,Y 338.96,Z 632.832,A -85,B 0,C 180,E1 -14221.188,E2 -14221.188} C_VEL
LIN {X 0,Y 338.972,Z 631.524,A -85,B 0,C 180,E1 -14222.377,E2 -14222.377} C_VEL
LIN {X 0,Y 339.128,Z 628.708,A -85,B 0,C 180,E1 -14224.16,E2 -14224.16} C_VEL
LIN {X 0,Y 339.212,Z 624.61,A -85,B 0,C 180,E1 -14226.007,E2 -14226.007} C_VEL
LIN {X 0,Y 339.418,Z 619.588,A -85,B 0,C 180,E1 -14227.735,E2 -14227.735} C_VEL
LIN {X 0,Y 339.773,Z 613.005,A -85,B 0,C 180,E1 -14229.525,E2 -14229.525} C_VEL
LIN {X 0,Y 340.312,Z 604.743,A -85,B 0,C 180,E1 -14231.314,E2 -14231.314} C_VEL
LIN {X 0,Y 340.996,Z 596.326,A -85,B 0,C 180,E1 -14232.801,E2 -14232.801} C_VEL
LIN {X 0,Y 341.772,Z 587.166,A -85,B 0,C 180,E1 -14234.134,E2 -14234.134} C_VEL
LIN {X 0,Y 342.483,Z 575.877,A -85,B 0,C 180,E1 -14235.472,E2 -14235.472} C_VEL
LIN {X 0,Y 343.163,Z 565.012,A -85,B 0,C 180,E1 -14236.509,E2 -14236.509} C_VEL
LIN {X 0,Y 343.909,Z 553.223,A -85,B 0,C 180,E1 -14237.39,E2 -14237.39} C_VEL
LIN {X 0,Y 344.595,Z 539.461,A -85,B 0,C 180,E1 -14238.159,E2 -14238.159} C_VEL
LIN {X 0,Y 345.133,Z 526.946,A -85,B 0,C 180,E1 -14238.63,E2 -14238.63} C_VEL
LIN {X 0,Y 347.203,Z 448.244,A -85,B 0,C 180,E1 -14240.84,E2 -14240.84} C_VEL
LIN {X 0,Y 344.071,Z 421.082,A -85,B 0,C 180,E1 -14241.769,E2 -14241.769} C_VEL
LIN {X 0,Y 344.076,Z 419.832,A -85,B 0,C 180,E1 -14241.887,E2 -14241.887} C_VEL
LIN {X 0,Y 345.416,Z 400.129,A -85,B 0,C 180,E1 -14245.295,E2 -14245.295} C_VEL
LIN {X 0,Y 346.614,Z 383.795,A -85,B 0,C 180,E1 -14248.127,E2 -14248.127} C_VEL
LIN {X 0,Y 345.587,Z 378.016,A -85,B 0,C 180,E1 -14249.214,E2 -14249.214} C_VEL
LIN {X 0,Y 341.386,Z 359.575,A -85,B 0,C 180,E1 -14252.807,E2 -14252.807} C_VEL
LIN {X 0,Y 340.762,Z 356.785,A -85,B 0,C 180,E1 -14253.417,E2 -14253.417} C_VEL
LIN {X 0,Y 340.71,Z 356.671,A -85,B 0,C 180,E1 -14256.741,E2 -14256.741} C_VEL
LIN {X 0,Y 340.694,Z 356.672,A -85,B 0,C 180,E1 -14260.246,E2 -14260.246} C_VEL
LIN {X 0,Y 340.657,Z 356.656,A -85,B 0,C 180,E1 -14263.772,E2 -14263.772} C_VEL
LIN {X 0,Y 340.705,Z 356.674,A -85,B 0,C 180,E1 -14267.954,E2 -14267.954} C_VEL
LIN {X 0,Y 340.741,Z 356.663,A -85,B 0,C 180,E1 -14271.772,E2 -14271.772} C_VEL
LIN {X 0,Y 340.728,Z 356.667,A -85,B 0,C 180,E1 -14275.595,E2 -14275.595} C_VEL
LIN {X 0,Y 340.769,Z 356.872,A -85,B 0,C 180,E1 -14276.958,E2 -14276.958} C_VEL
LIN {X 0,Y 343.873,Z 369.481,A -85,B 0,C 180,E1 -14280.625,E2 -14280.625} C_VEL
LIN {X 0,Y 344.51,Z 372.353,A -85,B 0,C 180,E1 -14281.345,E2 -14281.345} C_VEL
LIN {X 0,Y 352.15,Z 390.585,A -85,B 0,C 180,E1 -14282.463,E2 -14282.463} C_VEL
LIN {X 0,Y 355.841,Z 409.528,A -85,B 0,C 180,E1 -14283.194,E2 -14283.194} C_VEL
LIN {X 0,Y 353.545,Z 506.528,A -85,B 0,C 180,E1 -14285.168,E2 -14285.168} C_VEL
LIN {X 0,Y 352.777,Z 520.749,A -85,B 0,C 180,E1 -14285.621,E2 -14285.621} C_VEL
LIN {X 0,Y 351.81,Z 533.241,A -85,B 0,C 180,E1 -14286.215,E2 -14286.215} C_VEL
LIN {X 0,Y 350.621,Z 546.233,A -85,B 0,C 180,E1 -14287.053,E2 -14287.053} C_VEL
LIN {X 0,Y 349.261,Z 558.371,A -85,B 0,C 180,E1 -14288.058,E2 -14288.058} C_VEL
LIN {X 0,Y 347.736,Z 570.261,A -85,B 0,C 180,E1 -14289.286,E2 -14289.286} C_VEL
LIN {X 0,Y 346.054,Z 581.643,A -85,B 0,C 180,E1 -14290.729,E2 -14290.729} C_VEL
LIN {X 0,Y 344.592,Z 591.076,A -85,B 0,C 180,E1 -14292.185,E2 -14292.185} C_VEL
LIN {X 0,Y 343.092,Z 600.559,A -85,B 0,C 180,E1 -14293.945,E2 -14293.945} C_VEL
LIN {X 0,Y 341.951,Z 608.416,A -85,B 0,C 180,E1 -14295.72,E2 -14295.72} C_VEL
LIN {X 0,Y 340.973,Z 614.954,A -85,B 0,C 180,E1 -14297.5,E2 -14297.5} C_VEL
LIN {X 0,Y 340.24,Z 620.384,A -85,B 0,C 180,E1 -14299.285,E2 -14299.285} C_VEL
LIN {X 0,Y 339.527,Z 626.089,A -85,B 0,C 180,E1 -14301.667,E2 -14301.667} C_VEL
LIN {X 0,Y 339.191,Z 630.235,A -85,B 0,C 180,E1 -14304.052,E2 -14304.052} C_VEL
LIN {X 0,Y 339.061,Z 632.952,A -85,B 0,C 180,E1 -14306.433,E2 -14306.433} C_VEL
LIN {X 0,Y 338.955,Z 634.315,A -85,B 0,C 180,E1 -14308.81,E2 -14308.81} C_VEL
LIN {X 0,Y 338.955,Z 634.349,A -85,B 0,C 180,E1 -14311.187,E2 -14311.187} C_VEL
LIN {X 0,Y 339.058,Z 633.055,A -85,B 0,C 180,E1 -14313.564,E2 -14313.564} C_VEL
LIN {X 0,Y 339.207,Z 630.31,A -85,B 0,C 180,E1 -14316.005,E2 -14316.005} C_VEL
LIN {X 0,Y 339.523,Z 626.313,A -85,B 0,C 180,E1 -14318.33,E2 -14318.33} C_VEL
LIN {X 0,Y 340.183,Z 620.67,A -85,B 0,C 180,E1 -14320.714,E2 -14320.714} C_VEL
LIN {X 0,Y 341.127,Z 614.307,A -85,B 0,C 180,E1 -14322.794,E2 -14322.794} C_VEL
LIN {X 0,Y 341.388,Z 612.606,A -85,B 0,C 180,E1 -14323.284,E2 -14323.284} C_VEL
LIN {X 0,Y 341.213,Z 609.541,A -85,B 0,C 180,E1 -14324.132,E2 -14324.132} C_VEL
LIN {X 0,Y 339.156,Z 604.351,A -85,B 0,C 180,E1 -14325.516,E2 -14325.516} C_VEL
LIN {X 0,Y 337.205,Z 598.67,A -85,B 0,C 180,E1 -14326.855,E2 -14326.855} C_VEL
LIN {X 0,Y 337.191,Z 594.837,A -85,B 0,C 180,E1 -14327.619,E2 -14327.619} C_VEL
LIN {X 0,Y 338.902,Z 584.327,A -85,B 0,C 180,E1 -14329.376,E2 -14329.376} C_VEL
LIN {X 0,Y 340.607,Z 573.543,A -85,B 0,C 180,E1 -14330.849,E2 -14330.849} C_VEL
LIN {X 0,Y 342.307,Z 561.645,A -85,B 0,C 180,E1 -14332.174,E2 -14332.174} C_VEL
LIN {X 0,Y 343.866,Z 548.722,A -85,B 0,C 180,E1 -14333.326,E2 -14333.326} C_VEL
LIN {X 0,Y 345.205,Z 535.046,A -85,B 0,C 180,E1 -14334.266,E2 -14334.266} C_VEL
LIN {X 0,Y 346.407,Z 520.554,A -85,B 0,C 180,E1 -14334.975,E2 -14334.975} C_VEL
LIN {X 0,Y 347.123,Z 507.724,A -85,B 0,C 180,E1 -14335.4,E2 -14335.4} C_VEL
LIN {X 0,Y 349.568,Z 411.697,A -85,B 0,C 180,E1 -14337.387,E2 -14337.387} C_VEL
LIN {X 0,Y 347.755,Z 400.959,A -85,B 0,C 180,E1 -14337.787,E2 -14337.787} C_VEL
LIN {X 0,Y 345.674,Z 391.919,A -85,B 0,C 180,E1 -14338.178,E2 -14338.178} C_VEL
LIN {X 0,Y 337.372,Z 372.482,A -85,B 0,C 180,E1 -14339.425,E2 -14339.425} C_VEL
LIN {X 0,Y 336.72,Z 369.925,A -85,B 0,C 180,E1 -14340.059,E2 -14340.059} C_VEL
LIN {X 0,Y 333.717,Z 357.88,A -85,B 0,C 180,E1 -14343.649,E2 -14343.649} C_VEL
LIN {X 0,Y 333.657,Z 357.55,A -85,B 0,C 180,E1 -14343.928,E2 -14343.928} C_VEL
LIN {X 0,Y 333.653,Z 357.55,A -85,B 0,C 180,E1 -14347.649,E2 -14347.649} C_VEL
LIN {X 0,Y 333.694,Z 357.529,A -85,B 0,C 180,E1 -14350.758,E2 -14350.758} C_VEL
LIN {X 0,Y 333.724,Z 357.517,A -85,B 0,C 180,E1 -14354.273,E2 -14354.273} C_VEL
LIN {X 0,Y 333.699,Z 357.539,A -85,B 0,C 180,E1 -14357.627,E2 -14357.627} C_VEL
LIN {X 0,Y 333.675,Z 357.513,A -85,B 0,C 180,E1 -14361.194,E2 -14361.194} C_VEL
LIN {X 0,Y 333.677,Z 357.541,A -85,B 0,C 180,E1 -14365.225,E2 -14365.225} C_VEL
LIN {X 0,Y 333.626,Z 357.54,A -85,B 0,C 180,E1 -14368.221,E2 -14368.221} C_VEL
LIN {X 0,Y 333.702,Z 357.49,A -85,B 0,C 180,E1 -14371.027,E2 -14371.027} C_VEL
LIN {X 0,Y 333.726,Z 357.521,A -85,B 0,C 180,E1 -14373.753,E2 -14373.753} C_VEL
LIN {X 0,Y 333.71,Z 357.529,A -85,B 0,C 180,E1 -14377.913,E2 -14377.913} C_VEL
LIN {X 0,Y 333.784,Z 357.532,A -85,B 0,C 180,E1 -14381.589,E2 -14381.589} C_VEL
LIN {X 0,Y 333.798,Z 357.518,A -85,B 0,C 180,E1 -14385.576,E2 -14385.576} C_VEL
LIN {X 0,Y 333.828,Z 357.516,A -85,B 0,C 180,E1 -14389.078,E2 -14389.078} C_VEL
LIN {X 0,Y 334.015,Z 357.498,A -85,B 0,C 180,E1 -14392.747,E2 -14392.747} C_VEL
LIN {X 0,Y 333.805,Z 357.52,A -85,B 0,C 180,E1 -14395.169,E2 -14395.169} C_VEL
LIN {X 0,Y 334.098,Z 357.479,A -85,B 0,C 180,E1 -14397.589,E2 -14397.589} C_VEL
LIN {X 0,Y 334.278,Z 357.469,A -85,B 0,C 180,E1 -14400,E2 -14400} C_VEL
LIN {X 0,Y 334.098,Z 357.48,A -85,B 0,C 180,E1 -14402.411,E2 -14402.411} C_VEL
LIN {X 0,Y 334.015,Z 357.499,A -85,B 0,C 180,E1 -14407.253,E2 -14407.253} C_VEL
LIN {X 0,Y 333.827,Z 357.514,A -85,B 0,C 180,E1 -14410.922,E2 -14410.922} C_VEL
LIN {X 0,Y 333.798,Z 357.515,A -85,B 0,C 180,E1 -14414.635,E2 -14414.635} C_VEL
LIN {X 0,Y 333.786,Z 357.531,A -85,B 0,C 180,E1 -14418.656,E2 -14418.656} C_VEL
LIN {X 0,Y 333.682,Z 357.533,A -85,B 0,C 180,E1 -14422.279,E2 -14422.279} C_VEL
LIN {X 0,Y 333.72,Z 357.522,A -85,B 0,C 180,E1 -14426.248,E2 -14426.248} C_VEL
LIN {X 0,Y 333.672,Z 357.493,A -85,B 0,C 180,E1 -14428.976,E2 -14428.976} C_VEL
LIN {X 0,Y 333.629,Z 357.551,A -85,B 0,C 180,E1 -14433.209,E2 -14433.209} C_VEL
LIN {X 0,Y 333.657,Z 357.514,A -85,B 0,C 180,E1 -14436.834,E2 -14436.834} C_VEL
LIN {X 0,Y 333.691,Z 357.542,A -85,B 0,C 180,E1 -14440.761,E2 -14440.761} C_VEL
LIN {X 0,Y 333.723,Z 357.513,A -85,B 0,C 180,E1 -14444.276,E2 -14444.276} C_VEL
LIN {X 0,Y 333.7,Z 357.544,A -85,B 0,C 180,E1 -14447.63,E2 -14447.63} C_VEL
LIN {X 0,Y 333.677,Z 357.534,A -85,B 0,C 180,E1 -14451.197,E2 -14451.197} C_VEL
LIN {X 0,Y 333.68,Z 357.539,A -85,B 0,C 180,E1 -14455.227,E2 -14455.227} C_VEL
LIN {X 0,Y 333.692,Z 357.772,A -85,B 0,C 180,E1 -14456.348,E2 -14456.348} C_VEL
LIN {X 0,Y 336.429,Z 368.711,A -85,B 0,C 180,E1 -14459.636,E2 -14459.636} C_VEL
LIN {X 0,Y 337.293,Z 372.262,A -85,B 0,C 180,E1 -14460.595,E2 -14460.595} C_VEL
LIN {X 0,Y 344.561,Z 389.175,A -85,B 0,C 180,E1 -14461.705,E2 -14461.705} C_VEL
LIN {X 0,Y 346.332,Z 394.046,A -85,B 0,C 180,E1 -14461.975,E2 -14461.975} C_VEL
LIN {X 0,Y 349.581,Z 411.353,A -85,B 0,C 180,E1 -14462.651,E2 -14462.651} C_VEL
LIN {X 0,Y 347.108,Z 509.012,A -85,B 0,C 180,E1 -14464.679,E2 -14464.679} C_VEL
LIN {X 0,Y 346.184,Z 523.054,A -85,B 0,C 180,E1 -14465.168,E2 -14465.168} C_VEL
LIN {X 0,Y 345.028,Z 536.717,A -85,B 0,C 180,E1 -14465.881,E2 -14465.881} C_VEL
LIN {X 0,Y 343.741,Z 549.99,A -85,B 0,C 180,E1 -14466.825,E2 -14466.825} C_VEL
LIN {X 0,Y 342.292,Z 562.147,A -85,B 0,C 180,E1 -14467.926,E2 -14467.926} C_VEL
LIN {X 0,Y 340.502,Z 574.383,A -85,B 0,C 180,E1 -14469.303,E2 -14469.303} C_VEL
LIN {X 0,Y 338.636,Z 585.999,A -85,B 0,C 180,E1 -14470.923,E2 -14470.923} C_VEL
LIN {X 0,Y 336.933,Z 596.386,A -85,B 0,C 180,E1 -14472.71,E2 -14472.71} C_VEL
LIN {X 0,Y 335.417,Z 605.859,A -85,B 0,C 180,E1 -14474.729,E2 -14474.729} C_VEL
LIN {X 0,Y 334.362,Z 613.152,A -85,B 0,C 180,E1 -14476.633,E2 -14476.633} C_VEL
LIN {X 0,Y 333.381,Z 618.89,A -85,B 0,C 180,E1 -14478.449,E2 -14478.449} C_VEL
LIN {X 0,Y 332.779,Z 623.589,A -85,B 0,C 180,E1 -14480.275,E2 -14480.275} C_VEL
LIN {X 0,Y 332.269,Z 628.463,A -85,B 0,C 180,E1 -14482.711,E2 -14482.711} C_VEL
LIN {X 0,Y 332.023,Z 631.846,A -85,B 0,C 180,E1 -14485.145,E2 -14485.145} C_VEL
LIN {X 0,Y 331.885,Z 633.843,A -85,B 0,C 180,E1 -14487.574,E2 -14487.574} C_VEL
LIN {X 0,Y 331.855,Z 634.5,A -85,B 0,C 180,E1 -14490.002,E2 -14490.002} C_VEL
LIN {X 0,Y 331.886,Z 633.83,A -85,B 0,C 180,E1 -14492.429,E2 -14492.429} C_VEL
LIN {X 0,Y 332.014,Z 631.826,A -85,B 0,C 180,E1 -14494.859,E2 -14494.859} C_VEL
LIN {X 0,Y 332.257,Z 628.569,A -85,B 0,C 180,E1 -14497.293,E2 -14497.293} C_VEL
LIN {X 0,Y 332.645,Z 625.066,A -85,B 0,C 180,E1 -14499.119,E2 -14499.119} C_VEL
LIN {X 0,Y 333.383,Z 618.838,A -85,B 0,C 180,E1 -14501.554,E2 -14501.554} C_VEL
LIN {X 0,Y 334.546,Z 611.999,A -85,B 0,C 180,E1 -14503.672,E2 -14503.672} C_VEL
LIN {X 0,Y 335.748,Z 603.513,A -85,B 0,C 180,E1 -14505.792,E2 -14505.792} C_VEL
LIN {X 0,Y 337.192,Z 594.654,A -85,B 0,C 180,E1 -14507.592,E2 -14507.592} C_VEL
LIN {X 0,Y 338.945,Z 583.923,A -85,B 0,C 180,E1 -14509.377,E2 -14509.377} C_VEL
LIN {X 0,Y 340.666,Z 573.056,A -85,B 0,C 180,E1 -14510.848,E2 -14510.848} C_VEL
LIN {X 0,Y 342.372,Z 561.049,A -85,B 0,C 180,E1 -14512.173,E2 -14512.173} C_VEL
LIN {X 0,Y 343.694,Z 549.756,A -85,B 0,C 180,E1 -14513.182,E2 -14513.182} C_VEL
LIN {X 0,Y 345.044,Z 536.427,A -85,B 0,C 180,E1 -14514.121,E2 -14514.121} C_VEL
LIN {X 0,Y 346.193,Z 522.648,A -85,B 0,C 180,E1 -14514.834,E2 -14514.834} C_VEL
LIN {X 0,Y 347.04,Z 508.237,A -85,B 0,C 180,E1 -14515.33,E2 -14515.33} C_VEL
LIN {X 0,Y 349.237,Z 425.32,A -85,B 0,C 180,E1 -14517.069,E2 -14517.069} C_VEL
LIN {X 0,Y 350.294,Z 414.62,A -85,B 0,C 180,E1 -14517.482,E2 -14517.482} C_VEL
LIN {X 0,Y 351.126,Z 410.831,A -85,B 0,C 180,E1 -14517.767,E2 -14517.767} C_VEL
LIN {X 0,Y 352.079,Z 400.644,A -85,B 0,C 180,E1 -14518.847,E2 -14518.847} C_VEL
LIN {X 0,Y 351.901,Z 397.952,A -85,B 0,C 180,E1 -14519.25,E2 -14519.25} C_VEL
LIN {X 0,Y 349.656,Z 387.259,A -85,B 0,C 180,E1 -14521.508,E2 -14521.508} C_VEL
LIN {X 0,Y 349.018,Z 384.353,A -85,B 0,C 180,E1 -14522.249,E2 -14522.249} C_VEL
LIN {X 0,Y 346.9,Z 380.426,A -85,B 0,C 180,E1 -14523.836,E2 -14523.836} C_VEL
LIN {X 0,Y 345.116,Z 377.365,A -85,B 0,C 180,E1 -14525.456,E2 -14525.456} C_VEL
LIN {X 0,Y 343.073,Z 374.2,A -85,B 0,C 180,E1 -14527.922,E2 -14527.922} C_VEL
LIN {X 0,Y 342.415,Z 372.715,A -85,B 0,C 180,E1 -14529.516,E2 -14529.516} C_VEL
LIN {X 0,Y 341.988,Z 372.01,A -85,B 0,C 180,E1 -14531.12,E2 -14531.12} C_VEL
LIN {X 0,Y 341.839,Z 371.904,A -85,B 0,C 180,E1 -14532.725,E2 -14532.725} C_VEL
LIN {X 0,Y 341.857,Z 372.621,A -85,B 0,C 180,E1 -14534.347,E2 -14534.347} C_VEL
LIN {X 0,Y 342.886,Z 375.362,A -85,B 0,C 180,E1 -14537.553,E2 -14537.553} C_VEL
LIN {X 0,Y 344.23,Z 378.815,A -85,B 0,C 180,E1 -14539.948,E2 -14539.948} C_VEL
LIN {X 0,Y 345.933,Z 383.802,A -85,B 0,C 180,E1 -14542.448,E2 -14542.448} C_VEL
LIN {X 0,Y 347.685,Z 389.848,A -85,B 0,C 180,E1 -14544.819,E2 -14544.819} C_VEL
LIN {X 0,Y 349.192,Z 396.901,A -85,B 0,C 180,E1 -14547.084,E2 -14547.084} C_VEL
LIN {X 0,Y 349.98,Z 402.047,A -85,B 0,C 180,E1 -14548.526,E2 -14548.526} C_VEL
LIN {X 0,Y 349.902,Z 404.917,A -85,B 0,C 180,E1 -14549.191,E2 -14549.191} C_VEL
LIN {X 0,Y 347.401,Z 419.92,A -85,B 0,C 180,E1 -14552.066,E2 -14552.066} C_VEL
LIN {X 0,Y 350.517,Z 436.234,A -85,B 0,C 180,E1 -14553.456,E2 -14553.456} C_VEL
LIN {X 0,Y 352.509,Z 450.4,A -85,B 0,C 180,E1 -14554.443,E2 -14554.443} C_VEL
LIN {X 0,Y 352.75,Z 455.667,A -85,B 0,C 180,E1 -14554.722,E2 -14554.722} C_VEL
LIN {X 0,Y 347.008,Z 534.323,A -85,B 0,C 180,E1 -14557.407,E2 -14557.407} C_VEL
LIN {X 0,Y 345.567,Z 548.429,A -85,B 0,C 180,E1 -14558.134,E2 -14558.134} C_VEL
LIN {X 0,Y 343.987,Z 561.325,A -85,B 0,C 180,E1 -14559.051,E2 -14559.051} C_VEL
LIN {X 0,Y 342.237,Z 573.752,A -85,B 0,C 180,E1 -14560.194,E2 -14560.194} C_VEL
LIN {X 0,Y 340.448,Z 584.897,A -85,B 0,C 180,E1 -14561.495,E2 -14561.495} C_VEL
LIN {X 0,Y 338.75,Z 594.564,A -85,B 0,C 180,E1 -14562.875,E2 -14562.875} C_VEL
LIN {X 0,Y 337.256,Z 602.687,A -85,B 0,C 180,E1 -14564.282,E2 -14564.282} C_VEL
LIN {X 0,Y 335.765,Z 611.075,A -85,B 0,C 180,E1 -14566.072,E2 -14566.072} C_VEL
LIN {X 0,Y 334.672,Z 617.848,A -85,B 0,C 180,E1 -14567.878,E2 -14567.878} C_VEL
LIN {X 0,Y 333.634,Z 623.308,A -85,B 0,C 180,E1 -14569.686,E2 -14569.686} C_VEL
LIN {X 0,Y 332.83,Z 627.545,A -85,B 0,C 180,E1 -14571.5,E2 -14571.5} C_VEL
LIN {X 0,Y 332.356,Z 631.134,A -85,B 0,C 180,E1 -14573.657,E2 -14573.657} C_VEL
LIN {X 0,Y 332.151,Z 632.78,A -85,B 0,C 180,E1 -14575.145,E2 -14575.145} C_VEL
LIN {X 0,Y 332.022,Z 633.637,A -85,B 0,C 180,E1 -14576.359,E2 -14576.359} C_VEL
LIN {X 0,Y 331.905,Z 634.035,A -85,B 0,C 180,E1 -14577.573,E2 -14577.573} C_VEL
LIN {X 0,Y 331.871,Z 634.015,A -85,B 0,C 180,E1 -14578.787,E2 -14578.787} C_VEL
LIN {X 0,Y 331.86,Z 633.558,A -85,B 0,C 180,E1 -14580,E2 -14580} C_VEL
LIN {X 0,Y 331.869,Z 632.62,A -85,B 0,C 180,E1 -14581.214,E2 -14581.214} C_VEL
LIN {X 0,Y 331.893,Z 631.252,A -85,B 0,C 180,E1 -14582.427,E2 -14582.427} C_VEL
LIN {X 0,Y 332.041,Z 628.313,A -85,B 0,C 180,E1 -14584.249,E2 -14584.249} C_VEL
LIN {X 0,Y 332.145,Z 624.239,A -85,B 0,C 180,E1 -14586.073,E2 -14586.073} C_VEL
LIN {X 0,Y 332.414,Z 617.861,A -85,B 0,C 180,E1 -14588.205,E2 -14588.205} C_VEL
LIN {X 0,Y 332.849,Z 610.859,A -85,B 0,C 180,E1 -14590.032,E2 -14590.032} C_VEL
LIN {X 0,Y 333.318,Z 603.681,A -85,B 0,C 180,E1 -14591.555,E2 -14591.555} C_VEL
LIN {X 0,Y 333.998,Z 594.982,A -85,B 0,C 180,E1 -14593.074,E2 -14593.074} C_VEL
LIN {X 0,Y 334.83,Z 584.346,A -85,B 0,C 180,E1 -14594.589,E2 -14594.589} C_VEL
LIN {X 0,Y 335.564,Z 573.882,A -85,B 0,C 180,E1 -14595.8,E2 -14595.8} C_VEL
LIN {X 0,Y 336.471,Z 560.646,A -85,B 0,C 180,E1 -14597.003,E2 -14597.003} C_VEL
LIN {X 0,Y 337.227,Z 547.539,A -85,B 0,C 180,E1 -14597.903,E2 -14597.903} C_VEL
LIN {X 0,Y 337.913,Z 534.013,A -85,B 0,C 180,E1 -14598.571,E2 -14598.571} C_VEL
LIN {X 0,Y 338.705,Z 505.851,A -85,B 0,C 180,E1 -14599.429,E2 -14599.429} C_VEL
LIN {X 0,Y 340.276,Z 449.011,A -85,B 0,C 180,E1 -14601.08,E2 -14601.08} C_VEL
LIN {X 0,Y 337.188,Z 421.713,A -85,B 0,C 180,E1 -14602.035,E2 -14602.035} C_VEL
LIN {X 0,Y 337.122,Z 420.195,A -85,B 0,C 180,E1 -14602.12,E2 -14602.12} C_VEL
LIN {X 0,Y 338.608,Z 398.919,A -85,B 0,C 180,E1 -14605.841,E2 -14605.841} C_VEL
LIN {X 0,Y 339.617,Z 384.282,A -85,B 0,C 180,E1 -14608.422,E2 -14608.422} C_VEL
LIN {X 0,Y 336.17,Z 368.441,A -85,B 0,C 180,E1 -14611.511,E2 -14611.511} C_VEL
LIN {X 0,Y 333.72,Z 357.667,A -85,B 0,C 180,E1 -14613.719,E2 -14613.719} C_VEL
LIN {X 0,Y 333.657,Z 357.549,A -85,B 0,C 180,E1 -14617.651,E2 -14617.651} C_VEL
LIN {X 0,Y 333.652,Z 357.548,A -85,B 0,C 180,E1 -14620.767,E2 -14620.767} C_VEL
LIN {X 0,Y 333.598,Z 357.529,A -85,B 0,C 180,E1 -14624.25,E2 -14624.25} C_VEL
LIN {X 0,Y 333.647,Z 357.551,A -85,B 0,C 180,E1 -14627.618,E2 -14627.618} C_VEL
LIN {X 0,Y 333.659,Z 357.535,A -85,B 0,C 180,E1 -14631.201,E2 -14631.201} C_VEL
LIN {X 0,Y 333.683,Z 357.532,A -85,B 0,C 180,E1 -14633.86,E2 -14633.86} C_VEL
LIN {X 0,Y 333.677,Z 357.643,A -85,B 0,C 180,E1 -14636.343,E2 -14636.343} C_VEL
LIN {X 0,Y 336.105,Z 367.47,A -85,B 0,C 180,E1 -14639.342,E2 -14639.342} C_VEL
LIN {X 0,Y 337.304,Z 372.337,A -85,B 0,C 180,E1 -14640.671,E2 -14640.671} C_VEL
LIN {X 0,Y 345.766,Z 392.219,A -85,B 0,C 180,E1 -14641.948,E2 -14641.948} C_VEL
LIN {X 0,Y 347.128,Z 397.918,A -85,B 0,C 180,E1 -14642.198,E2 -14642.198} C_VEL
LIN {X 0,Y 349.54,Z 411.459,A -85,B 0,C 180,E1 -14642.714,E2 -14642.714} C_VEL
LIN {X 0,Y 347.015,Z 509.439,A -85,B 0,C 180,E1 -14644.748,E2 -14644.748} C_VEL
LIN {X 0,Y 346.085,Z 524.084,A -85,B 0,C 180,E1 -14645.278,E2 -14645.278} C_VEL
LIN {X 0,Y 345.014,Z 536.92,A -85,B 0,C 180,E1 -14645.957,E2 -14645.957} C_VEL
LIN {X 0,Y 343.729,Z 549.614,A -85,B 0,C 180,E1 -14646.853,E2 -14646.853} C_VEL
LIN {X 0,Y 342.288,Z 561.44,A -85,B 0,C 180,E1 -14647.91,E2 -14647.91} C_VEL
LIN {X 0,Y 340.567,Z 573.895,A -85,B 0,C 180,E1 -14649.304,E2 -14649.304} C_VEL
LIN {X 0,Y 338.997,Z 583.644,A -85,B 0,C 180,E1 -14650.626,E2 -14650.626} C_VEL
LIN {X 0,Y 337.247,Z 594.421,A -85,B 0,C 180,E1 -14652.411,E2 -14652.411} C_VEL
LIN {X 0,Y 335.752,Z 603.318,A -85,B 0,C 180,E1 -14654.208,E2 -14654.208} C_VEL
LIN {X 0,Y 334.562,Z 611.836,A -85,B 0,C 180,E1 -14656.329,E2 -14656.329} C_VEL
LIN {X 0,Y 333.408,Z 618.703,A -85,B 0,C 180,E1 -14658.447,E2 -14658.447} C_VEL
LIN {X 0,Y 332.79,Z 623.443,A -85,B 0,C 180,E1 -14660.272,E2 -14660.272} C_VEL
LIN {X 0,Y 332.259,Z 628.349,A -85,B 0,C 180,E1 -14662.707,E2 -14662.707} C_VEL
LIN {X 0,Y 332.019,Z 631.767,A -85,B 0,C 180,E1 -14665.141,E2 -14665.141} C_VEL
LIN {X 0,Y 331.887,Z 633.8,A -85,B 0,C 180,E1 -14667.571,E2 -14667.571} C_VEL
LIN {X 0,Y 331.856,Z 634.498,A -85,B 0,C 180,E1 -14669.998,E2 -14669.998} C_VEL
LIN {X 0,Y 331.886,Z 633.869,A -85,B 0,C 180,E1 -14672.426,E2 -14672.426} C_VEL
LIN {X 0,Y 332.014,Z 631.9,A -85,B 0,C 180,E1 -14674.856,E2 -14674.856} C_VEL
LIN {X 0,Y 332.269,Z 628.541,A -85,B 0,C 180,E1 -14677.289,E2 -14677.289} C_VEL
LIN {X 0,Y 332.778,Z 623.694,A -85,B 0,C 180,E1 -14679.725,E2 -14679.725} C_VEL
LIN {X 0,Y 333.627,Z 617.214,A -85,B 0,C 180,E1 -14682.159,E2 -14682.159} C_VEL
LIN {X 0,Y 334.815,Z 610,A -85,B 0,C 180,E1 -14684.277,E2 -14684.277} C_VEL
LIN {X 0,Y 336.227,Z 601.077,A -85,B 0,C 180,E1 -14686.389,E2 -14686.389} C_VEL
LIN {X 0,Y 337.191,Z 594.837,A -85,B 0,C 180,E1 -14687.619,E2 -14687.619} C_VEL
LIN {X 0,Y 337.239,Z 590.888,A -85,B 0,C 180,E1 -14688.36,E2 -14688.36} C_VEL
LIN {X 0,Y 335.608,Z 584.256,A -85,B 0,C 180,E1 -14689.586,E2 -14689.586} C_VEL
LIN {X 0,Y 334.009,Z 577.283,A -85,B 0,C 180,E1 -14690.76,E2 -14690.76} C_VEL
LIN {X 0,Y 334.077,Z 572.653,A -85,B 0,C 180,E1 -14691.398,E2 -14691.398} C_VEL
LIN {X 0,Y 335.898,Z 560.427,A -85,B 0,C 180,E1 -14692.758,E2 -14692.758} C_VEL
LIN {X 0,Y 337.362,Z 548.716,A -85,B 0,C 180,E1 -14693.803,E2 -14693.803} C_VEL
LIN {X 0,Y 338.73,Z 535.037,A -85,B 0,C 180,E1 -14694.76,E2 -14694.76} C_VEL
LIN {X 0,Y 339.985,Z 520.541,A -85,B 0,C 180,E1 -14695.48,E2 -14695.48} C_VEL
LIN {X 0,Y 340.72,Z 507.703,A -85,B 0,C 180,E1 -14695.913,E2 -14695.913} C_VEL
LIN {X 0,Y 343.241,Z 412.456,A -85,B 0,C 180,E1 -14697.918,E2 -14697.918} C_VEL
LIN {X 0,Y 340.974,Z 399.949,A -85,B 0,C 180,E1 -14698.413,E2 -14698.413} C_VEL
LIN {X 0,Y 339.821,Z 394.924,A -85,B 0,C 180,E1 -14698.636,E2 -14698.636} C_VEL
LIN {X 0,Y 332.584,Z 378.013,A -85,B 0,C 180,E1 -14699.729,E2 -14699.729} C_VEL
LIN {X 0,Y 330.018,Z 372.139,A -85,B 0,C 180,E1 -14700.181,E2 -14700.181} C_VEL
LIN {X 0,Y 327.335,Z 361.379,A -85,B 0,C 180,E1 -14703.388,E2 -14703.388} C_VEL
LIN {X 0,Y 326.643,Z 358.467,A -85,B 0,C 180,E1 -14704.385,E2 -14704.385} C_VEL
LIN {X 0,Y 326.643,Z 358.414,A -85,B 0,C 180,E1 -14708.603,E2 -14708.603} C_VEL
LIN {X 0,Y 326.625,Z 358.422,A -85,B 0,C 180,E1 -14711.836,E2 -14711.836} C_VEL
LIN {X 0,Y 326.665,Z 358.389,A -85,B 0,C 180,E1 -14715.23,E2 -14715.23} C_VEL
LIN {X 0,Y 326.625,Z 358.424,A -85,B 0,C 180,E1 -14718.856,E2 -14718.856} C_VEL
LIN {X 0,Y 326.639,Z 358.386,A -85,B 0,C 180,E1 -14721.393,E2 -14721.393} C_VEL
LIN {X 0,Y 326.612,Z 358.419,A -85,B 0,C 180,E1 -14724.85,E2 -14724.85} C_VEL
LIN {X 0,Y 326.601,Z 358.422,A -85,B 0,C 180,E1 -14727.455,E2 -14727.455} C_VEL
LIN {X 0,Y 326.652,Z 358.369,A -85,B 0,C 180,E1 -14730.34,E2 -14730.34} C_VEL
LIN {X 0,Y 326.681,Z 358.411,A -85,B 0,C 180,E1 -14734.515,E2 -14734.515} C_VEL
LIN {X 0,Y 326.636,Z 358.407,A -85,B 0,C 180,E1 -14738.544,E2 -14738.544} C_VEL
LIN {X 0,Y 326.734,Z 358.409,A -85,B 0,C 180,E1 -14741.177,E2 -14741.177} C_VEL
LIN {X 0,Y 326.752,Z 358.393,A -85,B 0,C 180,E1 -14745.433,E2 -14745.433} C_VEL
LIN {X 0,Y 326.763,Z 358.399,A -85,B 0,C 180,E1 -14748.839,E2 -14748.839} C_VEL
LIN {X 0,Y 326.969,Z 358.375,A -85,B 0,C 180,E1 -14752.59,E2 -14752.59} C_VEL
LIN {X 0,Y 326.771,Z 358.397,A -85,B 0,C 180,E1 -14755.065,E2 -14755.065} C_VEL
LIN {X 0,Y 327.039,Z 358.358,A -85,B 0,C 180,E1 -14757.537,E2 -14757.537} C_VEL
LIN {X 0,Y 327.229,Z 358.348,A -85,B 0,C 180,E1 -14760,E2 -14760} C_VEL
LIN {X 0,Y 327.039,Z 358.358,A -85,B 0,C 180,E1 -14762.463,E2 -14762.463} C_VEL
LIN {X 0,Y 326.987,Z 358.376,A -85,B 0,C 180,E1 -14766.169,E2 -14766.169} C_VEL
LIN {X 0,Y 326.904,Z 358.373,A -85,B 0,C 180,E1 -14768.655,E2 -14768.655} C_VEL
LIN {X 0,Y 326.729,Z 358.407,A -85,B 0,C 180,E1 -14772.421,E2 -14772.421} C_VEL
LIN {X 0,Y 326.743,Z 358.39,A -85,B 0,C 180,E1 -14774.958,E2 -14774.958} C_VEL
LIN {X 0,Y 326.723,Z 358.409,A -85,B 0,C 180,E1 -14778.839,E2 -14778.839} C_VEL
LIN {X 0,Y 326.613,Z 358.419,A -85,B 0,C 180,E1 -14782.788,E2 -14782.788} C_VEL
LIN {X 0,Y 326.679,Z 358.41,A -85,B 0,C 180,E1 -14785.485,E2 -14785.485} C_VEL
LIN {X 0,Y 326.635,Z 358.371,A -85,B 0,C 180,E1 -14788.253,E2 -14788.253} C_VEL
LIN {X 0,Y 326.565,Z 358.401,A -85,B 0,C 180,E1 -14791.098,E2 -14791.098} C_VEL
LIN {X 0,Y 326.599,Z 358.429,A -85,B 0,C 180,E1 -14794.02,E2 -14794.02} C_VEL
LIN {X 0,Y 326.621,Z 358.385,A -85,B 0,C 180,E1 -14797.24,E2 -14797.24} C_VEL
LIN {X 0,Y 326.627,Z 358.413,A -85,B 0,C 180,E1 -14800.204,E2 -14800.204} C_VEL
LIN {X 0,Y 326.651,Z 358.401,A -85,B 0,C 180,E1 -14803.511,E2 -14803.511} C_VEL
LIN {X 0,Y 326.644,Z 358.42,A -85,B 0,C 180,E1 -14807.015,E2 -14807.015} C_VEL
LIN {X 0,Y 326.639,Z 358.405,A -85,B 0,C 180,E1 -14810.767,E2 -14810.767} C_VEL
LIN {X 0,Y 326.607,Z 358.413,A -85,B 0,C 180,E1 -14814.482,E2 -14814.482} C_VEL
LIN {X 0,Y 326.648,Z 358.534,A -85,B 0,C 180,E1 -14815.708,E2 -14815.708} C_VEL
LIN {X 0,Y 328.99,Z 368.092,A -85,B 0,C 180,E1 -14818.704,E2 -14818.704} C_VEL
LIN {X 0,Y 330.023,Z 372.206,A -85,B 0,C 180,E1 -14819.873,E2 -14819.873} C_VEL
LIN {X 0,Y 335.852,Z 385.351,A -85,B 0,C 180,E1 -14820.809,E2 -14820.809} C_VEL
LIN {X 0,Y 340.162,Z 395.719,A -85,B 0,C 180,E1 -14821.459,E2 -14821.459} C_VEL
LIN {X 0,Y 343.27,Z 412.619,A -85,B 0,C 180,E1 -14822.134,E2 -14822.134} C_VEL
LIN {X 0,Y 340.713,Z 509.027,A -85,B 0,C 180,E1 -14824.169,E2 -14824.169} C_VEL
LIN {X 0,Y 339.709,Z 523.824,A -85,B 0,C 180,E1 -14824.703,E2 -14824.703} C_VEL
LIN {X 0,Y 338.438,Z 537.853,A -85,B 0,C 180,E1 -14825.462,E2 -14825.462} C_VEL
LIN {X 0,Y 337.001,Z 551.761,A -85,B 0,C 180,E1 -14826.496,E2 -14826.496} C_VEL
LIN {X 0,Y 335.546,Z 563.481,A -85,B 0,C 180,E1 -14827.61,E2 -14827.61} C_VEL
LIN {X 0,Y 333.649,Z 575.559,A -85,B 0,C 180,E1 -14829.019,E2 -14829.019} C_VEL
LIN {X 0,Y 331.896,Z 586.002,A -85,B 0,C 180,E1 -14830.52,E2 -14830.52} C_VEL
LIN {X 0,Y 330.117,Z 596.388,A -85,B 0,C 180,E1 -14832.341,E2 -14832.341} C_VEL
LIN {X 0,Y 328.63,Z 605.167,A -85,B 0,C 180,E1 -14834.23,E2 -14834.23} C_VEL
LIN {X 0,Y 327.441,Z 613.153,A -85,B 0,C 180,E1 -14836.345,E2 -14836.345} C_VEL
LIN {X 0,Y 326.39,Z 618.891,A -85,B 0,C 180,E1 -14838.198,E2 -14838.198} C_VEL
LIN {X 0,Y 325.764,Z 623.59,A -85,B 0,C 180,E1 -14840.063,E2 -14840.063} C_VEL
LIN {X 0,Y 325.197,Z 628.463,A -85,B 0,C 180,E1 -14842.551,E2 -14842.551} C_VEL
LIN {X 0,Y 325.059,Z 630.644,A -85,B 0,C 180,E1 -14844.016,E2 -14844.016} C_VEL
LIN {X 0,Y 324.877,Z 633.014,A -85,B 0,C 180,E1 -14846.281,E2 -14846.281} C_VEL
LIN {X 0,Y 324.775,Z 634.337,A -85,B 0,C 180,E1 -14848.762,E2 -14848.762} C_VEL
LIN {X 0,Y 324.775,Z 634.331,A -85,B 0,C 180,E1 -14851.242,E2 -14851.242} C_VEL
LIN {X 0,Y 324.875,Z 632.993,A -85,B 0,C 180,E1 -14853.723,E2 -14853.723} C_VEL
LIN {X 0,Y 325.074,Z 630.589,A -85,B 0,C 180,E1 -14856.207,E2 -14856.207} C_VEL
LIN {X 0,Y 325.334,Z 627.928,A -85,B 0,C 180,E1 -14858.073,E2 -14858.073} C_VEL
LIN {X 0,Y 325.8,Z 624.22,A -85,B 0,C 180,E1 -14859.939,E2 -14859.939} C_VEL
LIN {X 0,Y 326.448,Z 619.373,A -85,B 0,C 180,E1 -14861.803,E2 -14861.803} C_VEL
LIN {X 0,Y 327.625,Z 612.093,A -85,B 0,C 180,E1 -14863.966,E2 -14863.966} C_VEL
LIN {X 0,Y 328.877,Z 603.516,A -85,B 0,C 180,E1 -14866.131,E2 -14866.131} C_VEL
LIN {X 0,Y 330.408,Z 594.652,A -85,B 0,C 180,E1 -14867.966,E2 -14867.966} C_VEL
LIN {X 0,Y 332.248,Z 583.92,A -85,B 0,C 180,E1 -14869.784,E2 -14869.784} C_VEL
LIN {X 0,Y 333.999,Z 573.052,A -85,B 0,C 180,E1 -14871.284,E2 -14871.284} C_VEL
LIN {X 0,Y 335.737,Z 561.467,A -85,B 0,C 180,E1 -14872.587,E2 -14872.587} C_VEL
LIN {X 0,Y 337.172,Z 549.751,A -85,B 0,C 180,E1 -14873.658,E2 -14873.658} C_VEL
LIN {X 0,Y 338.582,Z 536.42,A -85,B 0,C 180,E1 -14874.611,E2 -14874.611} C_VEL
LIN {X 0,Y 339.78,Z 522.639,A -85,B 0,C 180,E1 -14875.336,E2 -14875.336} C_VEL
LIN {X 0,Y 340.658,Z 508.22,A -85,B 0,C 180,E1 -14875.839,E2 -14875.839} C_VEL
LIN {X 0,Y 342.418,Z 445.837,A -85,B 0,C 180,E1 -14877.174,E2 -14877.174} C_VEL
LIN {X 0,Y 345.609,Z 414.545,A -85,B 0,C 180,E1 -14878.371,E2 -14878.371} C_VEL
LIN {X 0,Y 346.203,Z 411.057,A -85,B 0,C 180,E1 -14878.692,E2 -14878.692} C_VEL
LIN {X 0,Y 347.133,Z 402.729,A -85,B 0,C 180,E1 -14879.632,E2 -14879.632} C_VEL
LIN {X 0,Y 345.046,Z 391.815,A -85,B 0,C 180,E1 -14881.978,E2 -14881.978} C_VEL
LIN {X 0,Y 344.542,Z 389.495,A -85,B 0,C 180,E1 -14882.598,E2 -14882.598} C_VEL
LIN {X 0,Y 342.672,Z 385.972,A -85,B 0,C 180,E1 -14884.048,E2 -14884.048} C_VEL
LIN {X 0,Y 340.264,Z 381.998,A -85,B 0,C 180,E1 -14886.339,E2 -14886.339} C_VEL
LIN {X 0,Y 338.735,Z 379.478,A -85,B 0,C 180,E1 -14888.496,E2 -14888.496} C_VEL
LIN {X 0,Y 338.11,Z 378.164,A -85,B 0,C 180,E1 -14890.12,E2 -14890.12} C_VEL
LIN {X 0,Y 337.705,Z 377.654,A -85,B 0,C 180,E1 -14891.757,E2 -14891.757} C_VEL
LIN {X 0,Y 337.554,Z 377.837,A -85,B 0,C 180,E1 -14893.4,E2 -14893.4} C_VEL
LIN {X 0,Y 337.57,Z 378.739,A -85,B 0,C 180,E1 -14895.063,E2 -14895.063} C_VEL
LIN {X 0,Y 337.985,Z 380.082,A -85,B 0,C 180,E1 -14896.703,E2 -14896.703} C_VEL
LIN {X 0,Y 338.726,Z 381.916,A -85,B 0,C 180,E1 -14898.398,E2 -14898.398} C_VEL
LIN {X 0,Y 340.016,Z 385.856,A -85,B 0,C 180,E1 -14900.856,E2 -14900.856} C_VEL
LIN {X 0,Y 341.639,Z 391.235,A -85,B 0,C 180,E1 -14903.375,E2 -14903.375} C_VEL
LIN {X 0,Y 342.899,Z 396.65,A -85,B 0,C 180,E1 -14905.392,E2 -14905.392} C_VEL
LIN {X 0,Y 344.124,Z 403.769,A -85,B 0,C 180,E1 -14907.625,E2 -14907.625} C_VEL
LIN {X 0,Y 344.267,Z 407.668,A -85,B 0,C 180,E1 -14908.63,E2 -14908.63} C_VEL
LIN {X 0,Y 342.023,Z 419.813,A -85,B 0,C 180,E1 -14911.022,E2 -14911.022} C_VEL
LIN {X 0,Y 344.637,Z 433.606,A -85,B 0,C 180,E1 -14912.313,E2 -14912.313} C_VEL
LIN {X 0,Y 346.857,Z 448.464,A -85,B 0,C 180,E1 -14913.472,E2 -14913.472} C_VEL
LIN {X 0,Y 347.483,Z 455.978,A -85,B 0,C 180,E1 -14913.943,E2 -14913.943} C_VEL
LIN {X 0,Y 341.329,Z 533.891,A -85,B 0,C 180,E1 -14916.689,E2 -14916.689} C_VEL
LIN {X 0,Y 339.768,Z 547.953,A -85,B 0,C 180,E1 -14917.421,E2 -14917.421} C_VEL
LIN {X 0,Y 338.322,Z 559.134,A -85,B 0,C 180,E1 -14918.203,E2 -14918.203} C_VEL
LIN {X 0,Y 336.412,Z 571.874,A -85,B 0,C 180,E1 -14919.358,E2 -14919.358} C_VEL
LIN {X 0,Y 334.488,Z 583.388,A -85,B 0,C 180,E1 -14920.675,E2 -14920.675} C_VEL
LIN {X 0,Y 332.386,Z 594.333,A -85,B 0,C 180,E1 -14922.243,E2 -14922.243} C_VEL
LIN {X 0,Y 330.524,Z 603.875,A -85,B 0,C 180,E1 -14923.953,E2 -14923.953} C_VEL
LIN {X 0,Y 328.946,Z 612.017,A -85,B 0,C 180,E1 -14925.777,E2 -14925.777} C_VEL
LIN {X 0,Y 327.781,Z 618.613,A -85,B 0,C 180,E1 -14927.619,E2 -14927.619} C_VEL
LIN {X 0,Y 326.684,Z 623.901,A -85,B 0,C 180,E1 -14929.464,E2 -14929.464} C_VEL
LIN {X 0,Y 325.825,Z 627.982,A -85,B 0,C 180,E1 -14931.316,E2 -14931.316} C_VEL
LIN {X 0,Y 325.275,Z 631.582,A -85,B 0,C 180,E1 -14933.672,E2 -14933.672} C_VEL
LIN {X 0,Y 325.08,Z 632.96,A -85,B 0,C 180,E1 -14935.039,E2 -14935.039} C_VEL
LIN {X 0,Y 324.935,Z 633.714,A -85,B 0,C 180,E1 -14936.28,E2 -14936.28} C_VEL
LIN {X 0,Y 324.827,Z 634.051,A -85,B 0,C 180,E1 -14937.52,E2 -14937.52} C_VEL
LIN {X 0,Y 324.783,Z 633.964,A -85,B 0,C 180,E1 -14938.76,E2 -14938.76} C_VEL
LIN {X 0,Y 324.77,Z 633.395,A -85,B 0,C 180,E1 -14940,E2 -14940} C_VEL
LIN {X 0,Y 324.78,Z 632.392,A -85,B 0,C 180,E1 -14941.24,E2 -14941.24} C_VEL
LIN {X 0,Y 324.816,Z 630.959,A -85,B 0,C 180,E1 -14942.48,E2 -14942.48} C_VEL
LIN {X 0,Y 324.955,Z 627.888,A -85,B 0,C 180,E1 -14944.341,E2 -14944.341} C_VEL
LIN {X 0,Y 325.061,Z 623.653,A -85,B 0,C 180,E1 -14946.206,E2 -14946.206} C_VEL
LIN {X 0,Y 325.379,Z 617.093,A -85,B 0,C 180,E1 -14948.384,E2 -14948.384} C_VEL
LIN {X 0,Y 325.805,Z 609.874,A -85,B 0,C 180,E1 -14950.251,E2 -14950.251} C_VEL
LIN {X 0,Y 326.446,Z 600.811,A -85,B 0,C 180,E1 -14952.117,E2 -14952.117} C_VEL
LIN {X 0,Y 327.09,Z 591.517,A -85,B 0,C 180,E1 -14953.671,E2 -14953.671} C_VEL
LIN {X 0,Y 327.787,Z 583.779,A -85,B 0,C 180,E1 -14954.751,E2 -14954.751} C_VEL
LIN {X 0,Y 328.573,Z 573.073,A -85,B 0,C 180,E1 -14955.995,E2 -14955.995} C_VEL
LIN {X 0,Y 329.377,Z 561.643,A -85,B 0,C 180,E1 -14957.061,E2 -14957.061} C_VEL
LIN {X 0,Y 330.096,Z 548.974,A -85,B 0,C 180,E1 -14957.982,E2 -14957.982} C_VEL
LIN {X 0,Y 330.831,Z 535.184,A -85,B 0,C 180,E1 -14958.702,E2 -14958.702} C_VEL
LIN {X 0,Y 331.265,Z 519.451,A -85,B 0,C 180,E1 -14959.239,E2 -14959.239} C_VEL
LIN {X 0,Y 333.323,Z 449.518,A -85,B 0,C 180,E1 -14961.326,E2 -14961.326} C_VEL
LIN {X 0,Y 330.298,Z 422.37,A -85,B 0,C 180,E1 -14962.296,E2 -14962.296} C_VEL
LIN {X 0,Y 330.178,Z 419.99,A -85,B 0,C 180,E1 -14962.439,E2 -14962.439} C_VEL
LIN {X 0,Y 331.677,Z 399.501,A -85,B 0,C 180,E1 -14966.083,E2 -14966.083} C_VEL
LIN {X 0,Y 332.708,Z 386.648,A -85,B 0,C 180,E1 -14968.378,E2 -14968.378} C_VEL
LIN {X 0,Y 331.539,Z 380.105,A -85,B 0,C 180,E1 -14969.641,E2 -14969.641} C_VEL
LIN {X 0,Y 327.531,Z 362.367,A -85,B 0,C 180,E1 -14973.19,E2 -14973.19} C_VEL
LIN {X 0,Y 326.668,Z 358.562,A -85,B 0,C 180,E1 -14974.012,E2 -14974.012} C_VEL
LIN {X 0,Y 326.633,Z 358.423,A -85,B 0,C 180,E1 -14977.238,E2 -14977.238} C_VEL
LIN {X 0,Y 326.584,Z 358.429,A -85,B 0,C 180,E1 -14981.131,E2 -14981.131} C_VEL
LIN {X 0,Y 326.532,Z 358.406,A -85,B 0,C 180,E1 -14984.742,E2 -14984.742} C_VEL
LIN {X 0,Y 326.582,Z 358.43,A -85,B 0,C 180,E1 -14988.153,E2 -14988.153} C_VEL
LIN {X 0,Y 326.63,Z 358.413,A -85,B 0,C 180,E1 -14991.391,E2 -14991.391} C_VEL
LIN {X 0,Y 326.644,Z 358.414,A -85,B 0,C 180,E1 -14995.236,E2 -14995.236} C_VEL
LIN {X 0,Y 326.665,Z 358.558,A -85,B 0,C 180,E1 -14995.8,E2 -14995.8} C_VEL
LIN {X 0,Y 329.326,Z 369.487,A -85,B 0,C 180,E1 -14999.19,E2 -14999.19} C_VEL
LIN {X 0,Y 330.119,Z 372.345,A -85,B 0,C 180,E1 -14999.968,E2 -14999.968} C_VEL
LIN {X 0,Y 339.021,Z 392.892,A -85,B 0,C 180,E1 -15001.354,E2 -15001.354} C_VEL
LIN {X 0,Y 340.325,Z 396.656,A -85,B 0,C 180,E1 -15001.562,E2 -15001.562} C_VEL
LIN {X 0,Y 343.198,Z 411.633,A -85,B 0,C 180,E1 -15002.17,E2 -15002.17} C_VEL
LIN {X 0,Y 340.815,Z 503.56,A -85,B 0,C 180,E1 -15004.092,E2 -15004.092} C_VEL
LIN {X 0,Y 340.076,Z 518.029,A -85,B 0,C 180,E1 -15004.524,E2 -15004.524} C_VEL
LIN {X 0,Y 338.974,Z 531.959,A -85,B 0,C 180,E1 -15005.174,E2 -15005.174} C_VEL
LIN {X 0,Y 337.646,Z 545.453,A -85,B 0,C 180,E1 -15006.052,E2 -15006.052} C_VEL
LIN {X 0,Y 336.074,Z 558.704,A -85,B 0,C 180,E1 -15007.182,E2 -15007.182} C_VEL
LIN {X 0,Y 334.265,Z 571.545,A -85,B 0,C 180,E1 -15008.572,E2 -15008.572} C_VEL
LIN {X 0,Y 332.626,Z 581.651,A -85,B 0,C 180,E1 -15009.918,E2 -15009.918} C_VEL
LIN {X 0,Y 331.066,Z 591.083,A -85,B 0,C 180,E1 -15011.431,E2 -15011.431} C_VEL
LIN {X 0,Y 329.388,Z 600.564,A -85,B 0,C 180,E1 -15013.258,E2 -15013.258} C_VEL
LIN {X 0,Y 328.084,Z 608.42,A -85,B 0,C 180,E1 -15015.103,E2 -15015.103} C_VEL
LIN {X 0,Y 327.09,Z 614.957,A -85,B 0,C 180,E1 -15016.96,E2 -15016.96} C_VEL
LIN {X 0,Y 326.198,Z 620.386,A -85,B 0,C 180,E1 -15018.818,E2 -15018.818} C_VEL
LIN {X 0,Y 325.437,Z 626.091,A -85,B 0,C 180,E1 -15021.304,E2 -15021.304} C_VEL
LIN {X 0,Y 325.055,Z 630.237,A -85,B 0,C 180,E1 -15023.792,E2 -15023.792} C_VEL
LIN {X 0,Y 324.878,Z 632.953,A -85,B 0,C 180,E1 -15026.277,E2 -15026.277} C_VEL
LIN {X 0,Y 324.776,Z 634.315,A -85,B 0,C 180,E1 -15028.758,E2 -15028.758} C_VEL
LIN {X 0,Y 324.775,Z 634.349,A -85,B 0,C 180,E1 -15031.238,E2 -15031.238} C_VEL
LIN {X 0,Y 324.875,Z 633.054,A -85,B 0,C 180,E1 -15033.719,E2 -15033.719} C_VEL
LIN {X 0,Y 325.053,Z 630.398,A -85,B 0,C 180,E1 -15036.204,E2 -15036.204} C_VEL
LIN {X 0,Y 325.432,Z 626.31,A -85,B 0,C 180,E1 -15038.693,E2 -15038.693} C_VEL
LIN {X 0,Y 326.15,Z 620.668,A -85,B 0,C 180,E1 -15041.181,E2 -15041.181} C_VEL
LIN {X 0,Y 327.214,Z 614.303,A -85,B 0,C 180,E1 -15043.348,E2 -15043.348} C_VEL
LIN {X 0,Y 328.459,Z 606.518,A -85,B 0,C 180,E1 -15045.478,E2 -15045.478} C_VEL
LIN {X 0,Y 329.847,Z 598.111,A -85,B 0,C 180,E1 -15047.353,E2 -15047.353} C_VEL
LIN {X 0,Y 331.538,Z 588.14,A -85,B 0,C 180,E1 -15049.18,E2 -15049.18} C_VEL
LIN {X 0,Y 333.418,Z 577.041,A -85,B 0,C 180,E1 -15050.835,E2 -15050.835} C_VEL
LIN {X 0,Y 334.077,Z 572.653,A -85,B 0,C 180,E1 -15051.398,E2 -15051.398} C_VEL
LIN {X 0,Y 334.179,Z 567.955,A -85,B 0,C 180,E1 -15052.015,E2 -15052.015} C_VEL
LIN {X 0,Y 332.683,Z 560.184,A -85,B 0,C 180,E1 -15053.044,E2 -15053.044} C_VEL
LIN {X 0,Y 331.115,Z 552.057,A -85,B 0,C 180,E1 -15053.984,E2 -15053.984} C_VEL
LIN {X 0,Y 331.087,Z 546.805,A -85,B 0,C 180,E1 -15054.451,E2 -15054.451} C_VEL
LIN {X 0,Y 332.445,Z 533.73,A -85,B 0,C 180,E1 -15055.345,E2 -15055.345} C_VEL
LIN {X 0,Y 333.656,Z 519.614,A -85,B 0,C 180,E1 -15056.041,E2 -15056.041} C_VEL
LIN {X 0,Y 334.41,Z 506.178,A -85,B 0,C 180,E1 -15056.481,E2 -15056.481} C_VEL
LIN {X 0,Y 336.97,Z 412.99,A -85,B 0,C 180,E1 -15058.471,E2 -15058.471} C_VEL
LIN {X 0,Y 333.97,Z 397.851,A -85,B 0,C 180,E1 -15059.114,E2 -15059.114} C_VEL
LIN {X 0,Y 326.184,Z 379.56,A -85,B 0,C 180,E1 -15060.334,E2 -15060.334} C_VEL
LIN {X 0,Y 322.794,Z 372.268,A -85,B 0,C 180,E1 -15060.912,E2 -15060.912} C_VEL
LIN {X 0,Y 320.205,Z 361.909,A -85,B 0,C 180,E1 -15064.079,E2 -15064.079} C_VEL
LIN {X 0,Y 319.601,Z 359.353,A -85,B 0,C 180,E1 -15064.994,E2 -15064.994} C_VEL
LIN {X 0,Y 319.595,Z 359.301,A -85,B 0,C 180,E1 -15068.002,E2 -15068.002} C_VEL
LIN {X 0,Y 319.597,Z 359.295,A -85,B 0,C 180,E1 -15071.611,E2 -15071.611} C_VEL
LIN {X 0,Y 319.639,Z 359.264,A -85,B 0,C 180,E1 -15075.284,E2 -15075.284} C_VEL
LIN {X 0,Y 319.582,Z 359.301,A -85,B 0,C 180,E1 -15078.72,E2 -15078.72} C_VEL
LIN {X 0,Y 319.575,Z 359.26,A -85,B 0,C 180,E1 -15082.342,E2 -15082.342} C_VEL
LIN {X 0,Y 319.552,Z 359.3,A -85,B 0,C 180,E1 -15085.122,E2 -15085.122} C_VEL
LIN {X 0,Y 319.562,Z 359.271,A -85,B 0,C 180,E1 -15089.057,E2 -15089.057} C_VEL
LIN {X 0,Y 319.599,Z 359.256,A -85,B 0,C 180,E1 -15092.497,E2 -15092.497} C_VEL
LIN {X 0,Y 319.597,Z 359.297,A -85,B 0,C 180,E1 -15095.303,E2 -15095.303} C_VEL
LIN {X 0,Y 319.587,Z 359.287,A -85,B 0,C 180,E1 -15098.047,E2 -15098.047} C_VEL
LIN {X 0,Y 319.679,Z 359.286,A -85,B 0,C 180,E1 -15100.961,E2 -15100.961} C_VEL
LIN {X 0,Y 319.72,Z 359.267,A -85,B 0,C 180,E1 -15105.275,E2 -15105.275} C_VEL
LIN {X 0,Y 319.749,Z 359.261,A -85,B 0,C 180,E1 -15109.872,E2 -15109.872} C_VEL
LIN {X 0,Y 319.923,Z 359.252,A -85,B 0,C 180,E1 -15112.426,E2 -15112.426} C_VEL
LIN {X 0,Y 319.74,Z 359.274,A -85,B 0,C 180,E1 -15114.956,E2 -15114.956} C_VEL
LIN {X 0,Y 319.982,Z 359.235,A -85,B 0,C 180,E1 -15117.482,E2 -15117.482} C_VEL
LIN {X 0,Y 320.179,Z 359.226,A -85,B 0,C 180,E1 -15120,E2 -15120} C_VEL
LIN {X 0,Y 319.982,Z 359.236,A -85,B 0,C 180,E1 -15122.518,E2 -15122.518} C_VEL
LIN {X 0,Y 319.942,Z 359.254,A -85,B 0,C 180,E1 -15126.306,E2 -15126.306} C_VEL
LIN {X 0,Y 319.832,Z 359.251,A -85,B 0,C 180,E1 -15128.848,E2 -15128.848} C_VEL
LIN {X 0,Y 319.675,Z 359.288,A -85,B 0,C 180,E1 -15132.7,E2 -15132.7} C_VEL
LIN {X 0,Y 319.689,Z 359.266,A -85,B 0,C 180,E1 -15135.296,E2 -15135.296} C_VEL
LIN {X 0,Y 319.664,Z 359.285,A -85,B 0,C 180,E1 -15139.256,E2 -15139.256} C_VEL
LIN {X 0,Y 319.562,Z 359.302,A -85,B 0,C 180,E1 -15143.32,E2 -15143.32} C_VEL
LIN {X 0,Y 319.605,Z 359.281,A -85,B 0,C 180,E1 -15146.091,E2 -15146.091} C_VEL
LIN {X 0,Y 319.558,Z 359.248,A -85,B 0,C 180,E1 -15148.937,E2 -15148.937} C_VEL
LIN {X 0,Y 319.516,Z 359.297,A -85,B 0,C 180,E1 -15151.864,E2 -15151.864} C_VEL
LIN {X 0,Y 319.571,Z 359.287,A -85,B 0,C 180,E1 -15155.544,E2 -15155.544} C_VEL
LIN {X 0,Y 319.575,Z 359.26,A -85,B 0,C 180,E1 -15158.008,E2 -15158.008} C_VEL
LIN {X 0,Y 319.61,Z 359.298,A -85,B 0,C 180,E1 -15161.617,E2 -15161.617} C_VEL
LIN {X 0,Y 319.639,Z 359.265,A -85,B 0,C 180,E1 -15165.287,E2 -15165.287} C_VEL
LIN {X 0,Y 319.577,Z 359.293,A -85,B 0,C 180,E1 -15168.722,E2 -15168.722} C_VEL
LIN {X 0,Y 319.593,Z 359.302,A -85,B 0,C 180,E1 -15172.341,E2 -15172.341} C_VEL
LIN {X 0,Y 319.619,Z 359.462,A -85,B 0,C 180,E1 -15175.133,E2 -15175.133} C_VEL
LIN {X 0,Y 322.164,Z 369.759,A -85,B 0,C 180,E1 -15178.431,E2 -15178.431} C_VEL
LIN {X 0,Y 322.845,Z 372.368,A -85,B 0,C 180,E1 -15179.148,E2 -15179.148} C_VEL
LIN {X 0,Y 330.539,Z 389.411,A -85,B 0,C 180,E1 -15180.393,E2 -15180.393} C_VEL
LIN {X 0,Y 334.219,Z 398.514,A -85,B 0,C 180,E1 -15180.97,E2 -15180.97} C_VEL
LIN {X 0,Y 336.976,Z 413.587,A -85,B 0,C 180,E1 -15181.589,E2 -15181.589} C_VEL
LIN {X 0,Y 334.738,Z 494.205,A -85,B 0,C 180,E1 -15183.295,E2 -15183.295} C_VEL
LIN {X 0,Y 334.133,Z 512.499,A -85,B 0,C 180,E1 -15183.747,E2 -15183.747} C_VEL
LIN {X 0,Y 333.081,Z 526.879,A -85,B 0,C 180,E1 -15184.331,E2 -15184.331} C_VEL
LIN {X 0,Y 331.777,Z 540.119,A -85,B 0,C 180,E1 -15185.104,E2 -15185.104} C_VEL
LIN {X 0,Y 330.258,Z 553.533,A -85,B 0,C 180,E1 -15186.153,E2 -15186.153} C_VEL
LIN {X 0,Y 328.668,Z 565.624,A -85,B 0,C 180,E1 -15187.364,E2 -15187.364} C_VEL
LIN {X 0,Y 326.633,Z 577.821,A -85,B 0,C 180,E1 -15188.877,E2 -15188.877} C_VEL
LIN {X 0,Y 324.886,Z 587.894,A -85,B 0,C 180,E1 -15190.411,E2 -15190.411} C_VEL
LIN {X 0,Y 323.048,Z 597.904,A -85,B 0,C 180,E1 -15192.269,E2 -15192.269} C_VEL
LIN {X 0,Y 321.5,Z 606.835,A -85,B 0,C 180,E1 -15194.308,E2 -15194.308} C_VEL
LIN {X 0,Y 320.307,Z 614.161,A -85,B 0,C 180,E1 -15196.359,E2 -15196.359} C_VEL
LIN {X 0,Y 319.145,Z 620.553,A -85,B 0,C 180,E1 -15198.57,E2 -15198.57} C_VEL
LIN {X 0,Y 318.383,Z 626.222,A -85,B 0,C 180,E1 -15201.113,E2 -15201.113} C_VEL
LIN {X 0,Y 317.971,Z 630.335,A -85,B 0,C 180,E1 -15203.657,E2 -15203.657} C_VEL
LIN {X 0,Y 317.79,Z 633.015,A -85,B 0,C 180,E1 -15206.198,E2 -15206.198} C_VEL
LIN {X 0,Y 317.689,Z 634.337,A -85,B 0,C 180,E1 -15208.734,E2 -15208.734} C_VEL
LIN {X 0,Y 317.689,Z 634.331,A -85,B 0,C 180,E1 -15211.269,E2 -15211.269} C_VEL
LIN {X 0,Y 317.788,Z 632.998,A -85,B 0,C 180,E1 -15213.806,E2 -15213.806} C_VEL
LIN {X 0,Y 318.008,Z 630.877,A -85,B 0,C 180,E1 -15216.346,E2 -15216.346} C_VEL
LIN {X 0,Y 318.325,Z 628.372,A -85,B 0,C 180,E1 -15218.252,E2 -15218.252} C_VEL
LIN {X 0,Y 318.827,Z 624.82,A -85,B 0,C 180,E1 -15220.159,E2 -15220.159} C_VEL
LIN {X 0,Y 319.545,Z 620.147,A -85,B 0,C 180,E1 -15222.062,E2 -15222.062} C_VEL
LIN {X 0,Y 320.822,Z 613.086,A -85,B 0,C 180,E1 -15224.269,E2 -15224.269} C_VEL
LIN {X 0,Y 321.806,Z 605.961,A -85,B 0,C 180,E1 -15226.069,E2 -15226.069} C_VEL
LIN {X 0,Y 323.345,Z 596.262,A -85,B 0,C 180,E1 -15228.044,E2 -15228.044} C_VEL
LIN {X 0,Y 325.195,Z 585.881,A -85,B 0,C 180,E1 -15229.902,E2 -15229.902} C_VEL
LIN {X 0,Y 327.211,Z 574.227,A -85,B 0,C 180,E1 -15231.583,E2 -15231.583} C_VEL
LIN {X 0,Y 329.123,Z 561.814,A -85,B 0,C 180,E1 -15233.026,E2 -15233.026} C_VEL
LIN {X 0,Y 330.679,Z 549.746,A -85,B 0,C 180,E1 -15234.151,E2 -15234.151} C_VEL
LIN {X 0,Y 332.117,Z 536.414,A -85,B 0,C 180,E1 -15235.123,E2 -15235.123} C_VEL
LIN {X 0,Y 333.379,Z 522.629,A -85,B 0,C 180,E1 -15235.858,E2 -15235.858} C_VEL
LIN {X 0,Y 334.283,Z 508.202,A -85,B 0,C 180,E1 -15236.369,E2 -15236.369} C_VEL
LIN {X 0,Y 335.642,Z 465.618,A -85,B 0,C 180,E1 -15237.304,E2 -15237.304} C_VEL
LIN {X 0,Y 340.999,Z 415.099,A -85,B 0,C 180,E1 -15239.266,E2 -15239.266} C_VEL
LIN {X 0,Y 342.028,Z 407.348,A -85,B 0,C 180,E1 -15240.129,E2 -15240.129} C_VEL
LIN {X 0,Y 342.096,Z 405.745,A -85,B 0,C 180,E1 -15240.362,E2 -15240.362} C_VEL
LIN {X 0,Y 340.467,Z 396.409,A -85,B 0,C 180,E1 -15242.461,E2 -15242.461} C_VEL
LIN {X 0,Y 340.13,Z 394.741,A -85,B 0,C 180,E1 -15242.913,E2 -15242.913} C_VEL
LIN {X 0,Y 338.066,Z 390.898,A -85,B 0,C 180,E1 -15244.587,E2 -15244.587} C_VEL
LIN {X 0,Y 336.351,Z 388.083,A -85,B 0,C 180,E1 -15246.227,E2 -15246.227} C_VEL
LIN {X 0,Y 334.383,Z 384.772,A -85,B 0,C 180,E1 -15249.091,E2 -15249.091} C_VEL
LIN {X 0,Y 333.794,Z 383.707,A -85,B 0,C 180,E1 -15250.747,E2 -15250.747} C_VEL
LIN {X 0,Y 333.39,Z 383.409,A -85,B 0,C 180,E1 -15252.454,E2 -15252.454} C_VEL
LIN {X 0,Y 333.204,Z 383.922,A -85,B 0,C 180,E1 -15254.182,E2 -15254.182} C_VEL
LIN {X 0,Y 333.346,Z 385.023,A -85,B 0,C 180,E1 -15255.913,E2 -15255.913} C_VEL
LIN {X 0,Y 333.848,Z 386.61,A -85,B 0,C 180,E1 -15257.651,E2 -15257.651} C_VEL
LIN {X 0,Y 334.944,Z 390.018,A -85,B 0,C 180,E1 -15260.146,E2 -15260.146} C_VEL
LIN {X 0,Y 336.269,Z 394.989,A -85,B 0,C 180,E1 -15262.692,E2 -15262.692} C_VEL
LIN {X 0,Y 337.425,Z 399.968,A -85,B 0,C 180,E1 -15264.722,E2 -15264.722} C_VEL
LIN {X 0,Y 338.622,Z 407.929,A -85,B 0,C 180,E1 -15267.342,E2 -15267.342} C_VEL
LIN {X 0,Y 338.685,Z 410.531,A -85,B 0,C 180,E1 -15268.053,E2 -15268.053} C_VEL
LIN {X 0,Y 336.851,Z 419.653,A -85,B 0,C 180,E1 -15269.901,E2 -15269.901} C_VEL
LIN {X 0,Y 339.218,Z 432.567,A -85,B 0,C 180,E1 -15271.219,E2 -15271.219} C_VEL
LIN {X 0,Y 341.411,Z 447.126,A -85,B 0,C 180,E1 -15272.463,E2 -15272.463} C_VEL
LIN {X 0,Y 342.303,Z 456.982,A -85,B 0,C 180,E1 -15273.148,E2 -15273.148} C_VEL
LIN {X 0,Y 335.642,Z 534.722,A -85,B 0,C 180,E1 -15275.983,E2 -15275.983} C_VEL
LIN {X 0,Y 333.93,Z 548.959,A -85,B 0,C 180,E1 -15276.758,E2 -15276.758} C_VEL
LIN {X 0,Y 332.25,Z 560.697,A -85,B 0,C 180,E1 -15277.62,E2 -15277.62} C_VEL
LIN {X 0,Y 330.245,Z 573.047,A -85,B 0,C 180,E1 -15278.791,E2 -15278.791} C_VEL
LIN {X 0,Y 328.203,Z 584.247,A -85,B 0,C 180,E1 -15280.127,E2 -15280.127} C_VEL
LIN {X 0,Y 326.176,Z 594.049,A -85,B 0,C 180,E1 -15281.564,E2 -15281.564} C_VEL
LIN {X 0,Y 324.191,Z 603.635,A -85,B 0,C 180,E1 -15283.307,E2 -15283.307} C_VEL
LIN {X 0,Y 322.357,Z 611.808,A -85,B 0,C 180,E1 -15285.157,E2 -15285.157} C_VEL
LIN {X 0,Y 321.251,Z 617.4,A -85,B 0,C 180,E1 -15286.72,E2 -15286.72} C_VEL
LIN {X 0,Y 320.05,Z 622.914,A -85,B 0,C 180,E1 -15288.602,E2 -15288.602} C_VEL
LIN {X 0,Y 319.11,Z 627.217,A -85,B 0,C 180,E1 -15290.492,E2 -15290.492} C_VEL
LIN {X 0,Y 318.45,Z 630.426,A -85,B 0,C 180,E1 -15292.391,E2 -15292.391} C_VEL
LIN {X 0,Y 318.162,Z 632.089,A -85,B 0,C 180,E1 -15293.742,E2 -15293.742} C_VEL
LIN {X 0,Y 317.995,Z 633.11,A -85,B 0,C 180,E1 -15294.928,E2 -15294.928} C_VEL
LIN {X 0,Y 317.851,Z 633.797,A -85,B 0,C 180,E1 -15296.197,E2 -15296.197} C_VEL
LIN {X 0,Y 317.752,Z 634.068,A -85,B 0,C 180,E1 -15297.465,E2 -15297.465} C_VEL
LIN {X 0,Y 317.698,Z 633.863,A -85,B 0,C 180,E1 -15298.733,E2 -15298.733} C_VEL
LIN {X 0,Y 317.683,Z 633.218,A -85,B 0,C 180,E1 -15300,E2 -15300} C_VEL
LIN {X 0,Y 317.695,Z 632.151,A -85,B 0,C 180,E1 -15301.268,E2 -15301.268} C_VEL
LIN {X 0,Y 317.796,Z 629.665,A -85,B 0,C 180,E1 -15303.169,E2 -15303.169} C_VEL
LIN {X 0,Y 317.846,Z 626.079,A -85,B 0,C 180,E1 -15305.074,E2 -15305.074} C_VEL
LIN {X 0,Y 318.099,Z 620.592,A -85,B 0,C 180,E1 -15307.209,E2 -15307.209} C_VEL
LIN {X 0,Y 318.457,Z 613.948,A -85,B 0,C 180,E1 -15309.207,E2 -15309.207} C_VEL
LIN {X 0,Y 318.942,Z 605.913,A -85,B 0,C 180,E1 -15311.117,E2 -15311.117} C_VEL
LIN {X 0,Y 319.756,Z 595.902,A -85,B 0,C 180,E1 -15313.02,E2 -15313.02} C_VEL
LIN {X 0,Y 320.55,Z 586.636,A -85,B 0,C 180,E1 -15314.442,E2 -15314.442} C_VEL
LIN {X 0,Y 321.331,Z 575.666,A -85,B 0,C 180,E1 -15315.821,E2 -15315.821} C_VEL
LIN {X 0,Y 322.114,Z 564.331,A -85,B 0,C 180,E1 -15316.967,E2 -15316.967} C_VEL
LIN {X 0,Y 322.901,Z 551.266,A -85,B 0,C 180,E1 -15317.987,E2 -15317.987} C_VEL
LIN {X 0,Y 323.659,Z 537.704,A -85,B 0,C 180,E1 -15318.762,E2 -15318.762} C_VEL
LIN {X 0,Y 324.17,Z 523.399,A -85,B 0,C 180,E1 -15319.307,E2 -15319.307} C_VEL
LIN {X 0,Y 326.384,Z 450.226,A -85,B 0,C 180,E1 -15321.571,E2 -15321.571} C_VEL
LIN {X 0,Y 323.419,Z 423.23,A -85,B 0,C 180,E1 -15322.562,E2 -15322.562} C_VEL
LIN {X 0,Y 323.233,Z 420.092,A -85,B 0,C 180,E1 -15322.715,E2 -15322.715} C_VEL
LIN {X 0,Y 324.742,Z 400.007,A -85,B 0,C 180,E1 -15326.338,E2 -15326.338} C_VEL
LIN {X 0,Y 325.699,Z 387.034,A -85,B 0,C 180,E1 -15328.693,E2 -15328.693} C_VEL
LIN {X 0,Y 322.695,Z 372.913,A -85,B 0,C 180,E1 -15331.514,E2 -15331.514} C_VEL
LIN {X 0,Y 319.631,Z 359.431,A -85,B 0,C 180,E1 -15334.34,E2 -15334.34} C_VEL
LIN {X 0,Y 319.563,Z 359.305,A -85,B 0,C 180,E1 -15338.01,E2 -15338.01} C_VEL
LIN {X 0,Y 319.531,Z 359.308,A -85,B 0,C 180,E1 -15341.596,E2 -15341.596} C_VEL
LIN {X 0,Y 319.493,Z 359.283,A -85,B 0,C 180,E1 -15345.256,E2 -15345.256} C_VEL
LIN {X 0,Y 319.534,Z 359.302,A -85,B 0,C 180,E1 -15348.711,E2 -15348.711} C_VEL
LIN {X 0,Y 319.584,Z 359.304,A -85,B 0,C 180,E1 -15352.343,E2 -15352.343} C_VEL
LIN {X 0,Y 319.648,Z 359.482,A -85,B 0,C 180,E1 -15355.225,E2 -15355.225} C_VEL
LIN {X 0,Y 322.115,Z 369.489,A -85,B 0,C 180,E1 -15358.422,E2 -15358.422} C_VEL
LIN {X 0,Y 322.809,Z 372.356,A -85,B 0,C 180,E1 -15359.216,E2 -15359.216} C_VEL
LIN {X 0,Y 328.512,Z 384.817,A -85,B 0,C 180,E1 -15360.147,E2 -15360.147} C_VEL
LIN {X 0,Y 334.244,Z 398.619,A -85,B 0,C 180,E1 -15361.043,E2 -15361.043} C_VEL
LIN {X 0,Y 336.927,Z 413.674,A -85,B 0,C 180,E1 -15361.653,E2 -15361.653} C_VEL
LIN {X 0,Y 334.296,Z 508.095,A -85,B 0,C 180,E1 -15363.674,E2 -15363.674} C_VEL
LIN {X 0,Y 333.377,Z 522.571,A -85,B 0,C 180,E1 -15364.184,E2 -15364.184} C_VEL
LIN {X 0,Y 332.213,Z 535.805,A -85,B 0,C 180,E1 -15364.884,E2 -15364.884} C_VEL
LIN {X 0,Y 330.747,Z 549.27,A -85,B 0,C 180,E1 -15365.854,E2 -15365.854} C_VEL
LIN {X 0,Y 329.211,Z 561.041,A -85,B 0,C 180,E1 -15366.936,E2 -15366.936} C_VEL
LIN {X 0,Y 327.475,Z 572.73,A -85,B 0,C 180,E1 -15368.27,E2 -15368.27} C_VEL
LIN {X 0,Y 325.598,Z 583.651,A -85,B 0,C 180,E1 -15369.795,E2 -15369.795} C_VEL
LIN {X 0,Y 323.688,Z 594.426,A -85,B 0,C 180,E1 -15371.648,E2 -15371.648} C_VEL
LIN {X 0,Y 322.034,Z 603.322,A -85,B 0,C 180,E1 -15373.517,E2 -15373.517} C_VEL
LIN {X 0,Y 320.881,Z 610.725,A -85,B 0,C 180,E1 -15375.41,E2 -15375.41} C_VEL
LIN {X 0,Y 319.757,Z 616.897,A -85,B 0,C 180,E1 -15377.302,E2 -15377.302} C_VEL
LIN {X 0,Y 318.758,Z 623.445,A -85,B 0,C 180,E1 -15379.839,E2 -15379.839} C_VEL
LIN {X 0,Y 318.13,Z 628.351,A -85,B 0,C 180,E1 -15382.382,E2 -15382.382} C_VEL
LIN {X 0,Y 317.848,Z 631.768,A -85,B 0,C 180,E1 -15384.924,E2 -15384.924} C_VEL
LIN {X 0,Y 317.732,Z 633.801,A -85,B 0,C 180,E1 -15387.463,E2 -15387.463} C_VEL
LIN {X 0,Y 317.679,Z 634.498,A -85,B 0,C 180,E1 -15389.998,E2 -15389.998} C_VEL
LIN {X 0,Y 317.731,Z 633.869,A -85,B 0,C 180,E1 -15392.534,E2 -15392.534} C_VEL
LIN {X 0,Y 317.842,Z 631.899,A -85,B 0,C 180,E1 -15395.073,E2 -15395.073} C_VEL
LIN {X 0,Y 318.132,Z 628.539,A -85,B 0,C 180,E1 -15397.615,E2 -15397.615} C_VEL
LIN {X 0,Y 318.736,Z 623.691,A -85,B 0,C 180,E1 -15400.158,E2 -15400.158} C_VEL
LIN {X 0,Y 319.731,Z 617.211,A -85,B 0,C 180,E1 -15402.696,E2 -15402.696} C_VEL
LIN {X 0,Y 320.818,Z 611.112,A -85,B 0,C 180,E1 -15404.59,E2 -15404.59} C_VEL
LIN {X 0,Y 322.283,Z 602.436,A -85,B 0,C 180,E1 -15406.793,E2 -15406.793} C_VEL
LIN {X 0,Y 323.914,Z 593.361,A -85,B 0,C 180,E1 -15408.663,E2 -15408.663} C_VEL
LIN {X 0,Y 325.864,Z 582.367,A -85,B 0,C 180,E1 -15410.514,E2 -15410.514} C_VEL
LIN {X 0,Y 327.719,Z 571.16,A -85,B 0,C 180,E1 -15412.04,E2 -15412.04} C_VEL
LIN {X 0,Y 329.56,Z 558.658,A -85,B 0,C 180,E1 -15413.411,E2 -15413.411} C_VEL
LIN {X 0,Y 331.087,Z 546.805,A -85,B 0,C 180,E1 -15414.451,E2 -15414.451} C_VEL
LIN {X 0,Y 331.118,Z 541.457,A -85,B 0,C 180,E1 -15414.895,E2 -15414.895} C_VEL
LIN {X 0,Y 329.371,Z 532.748,A -85,B 0,C 180,E1 -15415.662,E2 -15415.662} C_VEL
LIN {X 0,Y 327.586,Z 523.853,A -85,B 0,C 180,E1 -15416.348,E2 -15416.348} C_VEL
LIN {X 0,Y 327.362,Z 518.219,A -85,B 0,C 180,E1 -15416.645,E2 -15416.645} C_VEL
LIN {X 0,Y 328.156,Z 504.654,A -85,B 0,C 180,E1 -15417.07,E2 -15417.07} C_VEL
LIN {X 0,Y 330.72,Z 413.795,A -85,B 0,C 180,E1 -15419.04,E2 -15419.04} C_VEL
LIN {X 0,Y 328.03,Z 400.361,A -85,B 0,C 180,E1 -15419.631,E2 -15419.631} C_VEL
LIN {X 0,Y 320.514,Z 382.79,A -85,B 0,C 180,E1 -15420.846,E2 -15420.846} C_VEL
LIN {X 0,Y 315.561,Z 372.298,A -85,B 0,C 180,E1 -15421.697,E2 -15421.697} C_VEL
LIN {X 0,Y 313.017,Z 362.068,A -85,B 0,C 180,E1 -15424.925,E2 -15424.925} C_VEL
LIN {X 0,Y 312.554,Z 360.208,A -85,B 0,C 180,E1 -15425.65,E2 -15425.65} C_VEL
LIN {X 0,Y 312.533,Z 360.164,A -85,B 0,C 180,E1 -15429.021,E2 -15429.021} C_VEL
LIN {X 0,Y 312.556,Z 360.178,A -85,B 0,C 180,E1 -15432.418,E2 -15432.418} C_VEL
LIN {X 0,Y 312.586,Z 360.145,A -85,B 0,C 180,E1 -15436.008,E2 -15436.008} C_VEL
LIN {X 0,Y 312.541,Z 360.166,A -85,B 0,C 180,E1 -15439.863,E2 -15439.863} C_VEL
LIN {X 0,Y 312.533,Z 360.137,A -85,B 0,C 180,E1 -15442.616,E2 -15442.616} C_VEL
LIN {X 0,Y 312.511,Z 360.183,A -85,B 0,C 180,E1 -15446.31,E2 -15446.31} C_VEL
LIN {X 0,Y 312.536,Z 360.125,A -85,B 0,C 180,E1 -15450.349,E2 -15450.349} C_VEL
LIN {X 0,Y 312.593,Z 360.156,A -85,B 0,C 180,E1 -15454.063,E2 -15454.063} C_VEL
LIN {X 0,Y 312.578,Z 360.164,A -85,B 0,C 180,E1 -15457.528,E2 -15457.528} C_VEL
LIN {X 0,Y 312.628,Z 360.167,A -85,B 0,C 180,E1 -15461.656,E2 -15461.656} C_VEL
LIN {X 0,Y 312.684,Z 360.148,A -85,B 0,C 180,E1 -15465.686,E2 -15465.686} C_VEL
LIN {X 0,Y 312.693,Z 360.141,A -85,B 0,C 180,E1 -15469.641,E2 -15469.641} C_VEL
LIN {X 0,Y 312.861,Z 360.131,A -85,B 0,C 180,E1 -15472.254,E2 -15472.254} C_VEL
LIN {X 0,Y 312.711,Z 360.151,A -85,B 0,C 180,E1 -15474.842,E2 -15474.842} C_VEL
LIN {X 0,Y 312.985,Z 360.117,A -85,B 0,C 180,E1 -15478.713,E2 -15478.713} C_VEL
LIN {X 0,Y 313.131,Z 360.104,A -85,B 0,C 180,E1 -15480,E2 -15480} C_VEL
LIN {X 0,Y 312.929,Z 360.113,A -85,B 0,C 180,E1 -15482.574,E2 -15482.574} C_VEL
LIN {X 0,Y 312.9,Z 360.132,A -85,B 0,C 180,E1 -15486.448,E2 -15486.448} C_VEL
LIN {X 0,Y 312.777,Z 360.128,A -85,B 0,C 180,E1 -15489.049,E2 -15489.049} C_VEL
LIN {X 0,Y 312.627,Z 360.163,A -85,B 0,C 180,E1 -15492.991,E2 -15492.991} C_VEL
LIN {X 0,Y 312.628,Z 360.145,A -85,B 0,C 180,E1 -15495.65,E2 -15495.65} C_VEL
LIN {X 0,Y 312.62,Z 360.163,A -85,B 0,C 180,E1 -15499.237,E2 -15499.237} C_VEL
LIN {X 0,Y 312.537,Z 360.172,A -85,B 0,C 180,E1 -15502.79,E2 -15502.79} C_VEL
LIN {X 0,Y 312.585,Z 360.157,A -85,B 0,C 180,E1 -15505.934,E2 -15505.934} C_VEL
LIN {X 0,Y 312.498,Z 360.128,A -85,B 0,C 180,E1 -15509.655,E2 -15509.655} C_VEL
LIN {X 0,Y 312.51,Z 360.183,A -85,B 0,C 180,E1 -15513.69,E2 -15513.69} C_VEL
LIN {X 0,Y 312.533,Z 360.137,A -85,B 0,C 180,E1 -15517.384,E2 -15517.384} C_VEL
LIN {X 0,Y 312.531,Z 360.175,A -85,B 0,C 180,E1 -15520.703,E2 -15520.703} C_VEL
LIN {X 0,Y 312.588,Z 360.143,A -85,B 0,C 180,E1 -15524.185,E2 -15524.185} C_VEL
LIN {X 0,Y 312.55,Z 360.179,A -85,B 0,C 180,E1 -15527.905,E2 -15527.905} C_VEL
LIN {X 0,Y 312.553,Z 360.175,A -85,B 0,C 180,E1 -15531.906,E2 -15531.906} C_VEL
LIN {X 0,Y 312.559,Z 360.248,A -85,B 0,C 180,E1 -15534.424,E2 -15534.424} C_VEL
LIN {X 0,Y 314.319,Z 367.147,A -85,B 0,C 180,E1 -15536.786,E2 -15536.786} C_VEL
LIN {X 0,Y 315.544,Z 372.265,A -85,B 0,C 180,E1 -15538.342,E2 -15538.342} C_VEL
LIN {X 0,Y 322.154,Z 386.383,A -85,B 0,C 180,E1 -15539.464,E2 -15539.464} C_VEL
LIN {X 0,Y 328.284,Z 401.091,A -85,B 0,C 180,E1 -15540.457,E2 -15540.457} C_VEL
LIN {X 0,Y 330.745,Z 414.156,A -85,B 0,C 180,E1 -15541.016,E2 -15541.016} C_VEL
LIN {X 0,Y 328.425,Z 494.226,A -85,B 0,C 180,E1 -15542.739,E2 -15542.739} C_VEL
LIN {X 0,Y 327.79,Z 512.513,A -85,B 0,C 180,E1 -15543.199,E2 -15543.199} C_VEL
LIN {X 0,Y 326.683,Z 526.888,A -85,B 0,C 180,E1 -15543.79,E2 -15543.79} C_VEL
LIN {X 0,Y 325.235,Z 541.255,A -85,B 0,C 180,E1 -15544.653,E2 -15544.653} C_VEL
LIN {X 0,Y 323.587,Z 554.87,A -85,B 0,C 180,E1 -15545.767,E2 -15545.767} C_VEL
LIN {X 0,Y 321.89,Z 566.942,A -85,B 0,C 180,E1 -15547.03,E2 -15547.03} C_VEL
LIN {X 0,Y 319.811,Z 578.893,A -85,B 0,C 180,E1 -15548.573,E2 -15548.573} C_VEL
LIN {X 0,Y 317.849,Z 589.677,A -85,B 0,C 180,E1 -15550.296,E2 -15550.296} C_VEL
LIN {X 0,Y 315.986,Z 599.391,A -85,B 0,C 180,E1 -15552.194,E2 -15552.194} C_VEL
LIN {X 0,Y 314.546,Z 607.33,A -85,B 0,C 180,E1 -15554.085,E2 -15554.085} C_VEL
LIN {X 0,Y 313.396,Z 614.163,A -85,B 0,C 180,E1 -15556.052,E2 -15556.052} C_VEL
LIN {X 0,Y 312.143,Z 620.555,A -85,B 0,C 180,E1 -15558.311,E2 -15558.311} C_VEL
LIN {X 0,Y 311.355,Z 626.223,A -85,B 0,C 180,E1 -15560.911,E2 -15560.911} C_VEL
LIN {X 0,Y 310.899,Z 630.335,A -85,B 0,C 180,E1 -15563.512,E2 -15563.512} C_VEL
LIN {X 0,Y 310.706,Z 633.015,A -85,B 0,C 180,E1 -15566.111,E2 -15566.111} C_VEL
LIN {X 0,Y 310.606,Z 634.338,A -85,B 0,C 180,E1 -15568.705,E2 -15568.705} C_VEL
LIN {X 0,Y 310.606,Z 634.331,A -85,B 0,C 180,E1 -15571.298,E2 -15571.298} C_VEL
LIN {X 0,Y 310.704,Z 632.998,A -85,B 0,C 180,E1 -15573.893,E2 -15573.893} C_VEL
LIN {X 0,Y 310.958,Z 631.149,A -85,B 0,C 180,E1 -15576.49,E2 -15576.49} C_VEL
LIN {X 0,Y 311.149,Z 629.704,A -85,B 0,C 180,E1 -15577.79,E2 -15577.79} C_VEL
LIN {X 0,Y 311.654,Z 626.669,A -85,B 0,C 180,E1 -15579.739,E2 -15579.739} C_VEL
LIN {X 0,Y 312.332,Z 622.566,A -85,B 0,C 180,E1 -15581.686,E2 -15581.686} C_VEL
LIN {X 0,Y 313.589,Z 616.237,A -85,B 0,C 180,E1 -15583.943,E2 -15583.943} C_VEL
LIN {X 0,Y 314.844,Z 609.019,A -85,B 0,C 180,E1 -15585.989,E2 -15585.989} C_VEL
LIN {X 0,Y 316.195,Z 601.081,A -85,B 0,C 180,E1 -15587.797,E2 -15587.797} C_VEL
LIN {X 0,Y 317.944,Z 590.771,A -85,B 0,C 180,E1 -15589.701,E2 -15589.701} C_VEL
LIN {X 0,Y 319.812,Z 579.054,A -85,B 0,C 180,E1 -15591.43,E2 -15591.43} C_VEL
LIN {X 0,Y 322.287,Z 563.857,A -85,B 0,C 180,E1 -15593.303,E2 -15593.303} C_VEL
LIN {X 0,Y 323.971,Z 551.538,A -85,B 0,C 180,E1 -15594.514,E2 -15594.514} C_VEL
LIN {X 0,Y 325.57,Z 537.567,A -85,B 0,C 180,E1 -15595.579,E2 -15595.579} C_VEL
LIN {X 0,Y 326.94,Z 523.39,A -85,B 0,C 180,E1 -15596.363,E2 -15596.363} C_VEL
LIN {X 0,Y 327.901,Z 509.543,A -85,B 0,C 180,E1 -15596.881,E2 -15596.881} C_VEL
LIN {X 0,Y 328.866,Z 484.525,A -85,B 0,C 180,E1 -15597.483,E2 -15597.483} C_VEL
LIN {X 0,Y 336.288,Z 417.694,A -85,B 0,C 180,E1 -15600.105,E2 -15600.105} C_VEL
LIN {X 0,Y 336.524,Z 414.771,A -85,B 0,C 180,E1 -15600.326,E2 -15600.326} C_VEL
LIN {X 0,Y 337.217,Z 410.377,A -85,B 0,C 180,E1 -15600.849,E2 -15600.849} C_VEL
LIN {X 0,Y 336.632,Z 406.275,A -85,B 0,C 180,E1 -15601.71,E2 -15601.71} C_VEL
LIN {X 0,Y 335.773,Z 400.321,A -85,B 0,C 180,E1 -15603.151,E2 -15603.151} C_VEL
LIN {X 0,Y 334.086,Z 396.849,A -85,B 0,C 180,E1 -15604.611,E2 -15604.611} C_VEL
LIN {X 0,Y 332.14,Z 393.665,A -85,B 0,C 180,E1 -15606.479,E2 -15606.479} C_VEL
LIN {X 0,Y 330.822,Z 391.557,A -85,B 0,C 180,E1 -15608.184,E2 -15608.184} C_VEL
LIN {X 0,Y 329.937,Z 390.03,A -85,B 0,C 180,E1 -15609.929,E2 -15609.929} C_VEL
LIN {X 0,Y 329.366,Z 389.253,A -85,B 0,C 180,E1 -15611.684,E2 -15611.684} C_VEL
LIN {X 0,Y 329.019,Z 389.35,A -85,B 0,C 180,E1 -15613.427,E2 -15613.427} C_VEL
LIN {X 0,Y 328.913,Z 390.15,A -85,B 0,C 180,E1 -15615.161,E2 -15615.161} C_VEL
LIN {X 0,Y 329.163,Z 391.47,A -85,B 0,C 180,E1 -15616.903,E2 -15616.903} C_VEL
LIN {X 0,Y 329.686,Z 393.344,A -85,B 0,C 180,E1 -15618.637,E2 -15618.637} C_VEL
LIN {X 0,Y 330.646,Z 397.05,A -85,B 0,C 180,E1 -15621.034,E2 -15621.034} C_VEL
LIN {X 0,Y 331.871,Z 402.49,A -85,B 0,C 180,E1 -15623.633,E2 -15623.633} C_VEL
LIN {X 0,Y 332.649,Z 407.399,A -85,B 0,C 180,E1 -15625.486,E2 -15625.486} C_VEL
LIN {X 0,Y 333.185,Z 412.478,A -85,B 0,C 180,E1 -15627.138,E2 -15627.138} C_VEL
LIN {X 0,Y 332.992,Z 415.059,A -85,B 0,C 180,E1 -15627.797,E2 -15627.797} C_VEL
LIN {X 0,Y 332.023,Z 419.74,A -85,B 0,C 180,E1 -15628.735,E2 -15628.735} C_VEL
LIN {X 0,Y 334.385,Z 433.601,A -85,B 0,C 180,E1 -15630.252,E2 -15630.252} C_VEL
LIN {X 0,Y 336.415,Z 448.191,A -85,B 0,C 180,E1 -15631.577,E2 -15631.577} C_VEL
LIN {X 0,Y 337.273,Z 458.426,A -85,B 0,C 180,E1 -15632.333,E2 -15632.333} C_VEL
LIN {X 0,Y 330.205,Z 534.487,A -85,B 0,C 180,E1 -15635.185,E2 -15635.185} C_VEL
LIN {X 0,Y 328.303,Z 549.177,A -85,B 0,C 180,E1 -15636,E2 -15636} C_VEL
LIN {X 0,Y 326.248,Z 562.433,A -85,B 0,C 180,E1 -15637.018,E2 -15637.018} C_VEL
LIN {X 0,Y 324.147,Z 574.369,A -85,B 0,C 180,E1 -15638.204,E2 -15638.204} C_VEL
LIN {X 0,Y 321.721,Z 586.46,A -85,B 0,C 180,E1 -15639.726,E2 -15639.726} C_VEL
LIN {X 0,Y 319.314,Z 597.094,A -85,B 0,C 180,E1 -15641.407,E2 -15641.407} C_VEL
LIN {X 0,Y 317.126,Z 606.433,A -85,B 0,C 180,E1 -15643.256,E2 -15643.256} C_VEL
LIN {X 0,Y 315.348,Z 614.039,A -85,B 0,C 180,E1 -15645.15,E2 -15645.15} C_VEL
LIN {X 0,Y 314.029,Z 620.18,A -85,B 0,C 180,E1 -15647.068,E2 -15647.068} C_VEL
LIN {X 0,Y 312.783,Z 625.091,A -85,B 0,C 180,E1 -15648.99,E2 -15648.99} C_VEL
LIN {X 0,Y 311.831,Z 628.859,A -85,B 0,C 180,E1 -15650.923,E2 -15650.923} C_VEL
LIN {X 0,Y 311.42,Z 630.796,A -85,B 0,C 180,E1 -15652.218,E2 -15652.218} C_VEL
LIN {X 0,Y 311.083,Z 632.463,A -85,B 0,C 180,E1 -15653.757,E2 -15653.757} C_VEL
LIN {X 0,Y 310.77,Z 633.886,A -85,B 0,C 180,E1 -15656.11,E2 -15656.11} C_VEL
LIN {X 0,Y 310.678,Z 634.038,A -85,B 0,C 180,E1 -15657.407,E2 -15657.407} C_VEL
LIN {X 0,Y 310.615,Z 633.744,A -85,B 0,C 180,E1 -15658.704,E2 -15658.704} C_VEL
LIN {X 0,Y 310.597,Z 633.031,A -85,B 0,C 180,E1 -15660,E2 -15660} C_VEL
LIN {X 0,Y 310.612,Z 631.862,A -85,B 0,C 180,E1 -15661.297,E2 -15661.297} C_VEL
LIN {X 0,Y 310.731,Z 629.235,A -85,B 0,C 180,E1 -15663.242,E2 -15663.242} C_VEL
LIN {X 0,Y 310.767,Z 625.474,A -85,B 0,C 180,E1 -15665.19,E2 -15665.19} C_VEL
LIN {X 0,Y 311.017,Z 620.223,A -85,B 0,C 180,E1 -15667.232,E2 -15667.232} C_VEL
LIN {X 0,Y 311.362,Z 614.162,A -85,B 0,C 180,E1 -15669.091,E2 -15669.091} C_VEL
LIN {X 0,Y 311.824,Z 606.196,A -85,B 0,C 180,E1 -15671.045,E2 -15671.045} C_VEL
LIN {X 0,Y 312.632,Z 596.248,A -85,B 0,C 180,E1 -15672.991,E2 -15672.991} C_VEL
LIN {X 0,Y 313.404,Z 587.061,A -85,B 0,C 180,E1 -15674.447,E2 -15674.447} C_VEL
LIN {X 0,Y 314.275,Z 575.56,A -85,B 0,C 180,E1 -15675.927,E2 -15675.927} C_VEL
LIN {X 0,Y 315.149,Z 563.2,A -85,B 0,C 180,E1 -15677.187,E2 -15677.187} C_VEL
LIN {X 0,Y 315.964,Z 549.921,A -85,B 0,C 180,E1 -15678.228,E2 -15678.228} C_VEL
LIN {X 0,Y 316.737,Z 535.8,A -85,B 0,C 180,E1 -15679.02,E2 -15679.02} C_VEL
LIN {X 0,Y 317.197,Z 522.002,A -85,B 0,C 180,E1 -15679.538,E2 -15679.538} C_VEL
LIN {X 0,Y 319.436,Z 450.881,A -85,B 0,C 180,E1 -15681.813,E2 -15681.813} C_VEL
LIN {X 0,Y 316.533,Z 423.937,A -85,B 0,C 180,E1 -15682.831,E2 -15682.831} C_VEL
LIN {X 0,Y 316.265,Z 420.16,A -85,B 0,C 180,E1 -15683.006,E2 -15683.006} C_VEL
LIN {X 0,Y 317.814,Z 400.455,A -85,B 0,C 180,E1 -15686.603,E2 -15686.603} C_VEL
LIN {X 0,Y 318.747,Z 389.086,A -85,B 0,C 180,E1 -15688.695,E2 -15688.695} C_VEL
LIN {X 0,Y 317.856,Z 383.731,A -85,B 0,C 180,E1 -15689.758,E2 -15689.758} C_VEL
LIN {X 0,Y 314.032,Z 366.73,A -85,B 0,C 180,E1 -15693.251,E2 -15693.251} C_VEL
LIN {X 0,Y 312.576,Z 360.307,A -85,B 0,C 180,E1 -15694.665,E2 -15694.665} C_VEL
LIN {X 0,Y 312.511,Z 360.184,A -85,B 0,C 180,E1 -15698.082,E2 -15698.082} C_VEL
LIN {X 0,Y 312.49,Z 360.185,A -85,B 0,C 180,E1 -15702.081,E2 -15702.081} C_VEL
LIN {X 0,Y 312.463,Z 360.165,A -85,B 0,C 180,E1 -15706.034,E2 -15706.034} C_VEL
LIN {X 0,Y 312.51,Z 360.163,A -85,B 0,C 180,E1 -15709.874,E2 -15709.874} C_VEL
LIN {X 0,Y 312.544,Z 360.178,A -85,B 0,C 180,E1 -15712.616,E2 -15712.616} C_VEL
LIN {X 0,Y 312.558,Z 360.274,A -85,B 0,C 180,E1 -15714.519,E2 -15714.519} C_VEL
LIN {X 0,Y 314.876,Z 369.492,A -85,B 0,C 180,E1 -15717.609,E2 -15717.609} C_VEL
LIN {X 0,Y 315.631,Z 372.528,A -85,B 0,C 180,E1 -15718.453,E2 -15718.453} C_VEL
LIN {X 0,Y 322.904,Z 388.183,A -85,B 0,C 180,E1 -15719.659,E2 -15719.659} C_VEL
LIN {X 0,Y 328.362,Z 401.49,A -85,B 0,C 180,E1 -15720.543,E2 -15720.543} C_VEL
LIN {X 0,Y 330.682,Z 414.453,A -85,B 0,C 180,E1 -15721.086,E2 -15721.086} C_VEL
LIN {X 0,Y 328.271,Z 498.421,A -85,B 0,C 180,E1 -15722.894,E2 -15722.894} C_VEL
LIN {X 0,Y 327.659,Z 514.052,A -85,B 0,C 180,E1 -15723.313,E2 -15723.313} C_VEL
LIN {X 0,Y 326.534,Z 527.926,A -85,B 0,C 180,E1 -15723.902,E2 -15723.902} C_VEL
LIN {X 0,Y 325.169,Z 541.456,A -85,B 0,C 180,E1 -15724.73,E2 -15724.73} C_VEL
LIN {X 0,Y 323.466,Z 555.185,A -85,B 0,C 180,E1 -15725.859,E2 -15725.859} C_VEL
LIN {X 0,Y 321.691,Z 567.697,A -85,B 0,C 180,E1 -15727.182,E2 -15727.182} C_VEL
LIN {X 0,Y 319.647,Z 579.52,A -85,B 0,C 180,E1 -15728.727,E2 -15728.727} C_VEL
LIN {X 0,Y 317.876,Z 589.308,A -85,B 0,C 180,E1 -15730.294,E2 -15730.294} C_VEL
LIN {X 0,Y 316.013,Z 599.084,A -85,B 0,C 180,E1 -15732.193,E2 -15732.193} C_VEL
LIN {X 0,Y 314.537,Z 607.113,A -85,B 0,C 180,E1 -15734.091,E2 -15734.091} C_VEL
LIN {X 0,Y 313.405,Z 613.954,A -85,B 0,C 180,E1 -15736.049,E2 -15736.049} C_VEL
LIN {X 0,Y 312.175,Z 620.389,A -85,B 0,C 180,E1 -15738.308,E2 -15738.308} C_VEL
LIN {X 0,Y 311.361,Z 626.094,A -85,B 0,C 180,E1 -15740.907,E2 -15740.907} C_VEL
LIN {X 0,Y 310.902,Z 630.238,A -85,B 0,C 180,E1 -15743.509,E2 -15743.509} C_VEL
LIN {X 0,Y 310.706,Z 632.954,A -85,B 0,C 180,E1 -15746.107,E2 -15746.107} C_VEL
LIN {X 0,Y 310.607,Z 634.316,A -85,B 0,C 180,E1 -15748.702,E2 -15748.702} C_VEL
LIN {X 0,Y 310.607,Z 634.349,A -85,B 0,C 180,E1 -15751.295,E2 -15751.295} C_VEL
LIN {X 0,Y 310.703,Z 633.053,A -85,B 0,C 180,E1 -15753.889,E2 -15753.889} C_VEL
LIN {X 0,Y 310.9,Z 630.397,A -85,B 0,C 180,E1 -15756.488,E2 -15756.488} C_VEL
LIN {X 0,Y 311.355,Z 626.308,A -85,B 0,C 180,E1 -15759.089,E2 -15759.089} C_VEL
LIN {X 0,Y 312.132,Z 620.665,A -85,B 0,C 180,E1 -15761.69,E2 -15761.69} C_VEL
LIN {X 0,Y 313.371,Z 614.3,A -85,B 0,C 180,E1 -15763.949,E2 -15763.949} C_VEL
LIN {X 0,Y 314.735,Z 606.328,A -85,B 0,C 180,E1 -15766.221,E2 -15766.221} C_VEL
LIN {X 0,Y 316.238,Z 598.106,A -85,B 0,C 180,E1 -15768.126,E2 -15768.126} C_VEL
LIN {X 0,Y 318.094,Z 588.134,A -85,B 0,C 180,E1 -15770.025,E2 -15770.025} C_VEL
LIN {X 0,Y 320.153,Z 577.034,A -85,B 0,C 180,E1 -15771.741,E2 -15771.741} C_VEL
LIN {X 0,Y 321.996,Z 565.988,A -85,B 0,C 180,E1 -15773.131,E2 -15773.131} C_VEL
LIN {X 0,Y 323.733,Z 553.994,A -85,B 0,C 180,E1 -15774.359,E2 -15774.359} C_VEL
LIN {X 0,Y 325.321,Z 540.719,A -85,B 0,C 180,E1 -15775.425,E2 -15775.425} C_VEL
LIN {X 0,Y 326.68,Z 526.924,A -85,B 0,C 180,E1 -15776.253,E2 -15776.253} C_VEL
LIN {X 0,Y 327.362,Z 518.219,A -85,B 0,C 180,E1 -15776.645,E2 -15776.645} C_VEL
LIN {X 0,Y 327.127,Z 512.504,A -85,B 0,C 180,E1 -15776.908,E2 -15776.908} C_VEL
LIN {X 0,Y 322.79,Z 493.871,A -85,B 0,C 180,E1 -15777.836,E2 -15777.836} C_VEL
LIN {X 0,Y 322.395,Z 488.057,A -85,B 0,C 180,E1 -15778.012,E2 -15778.012} C_VEL
LIN {X 0,Y 324.442,Z 414.593,A -85,B 0,C 180,E1 -15779.637,E2 -15779.637} C_VEL
LIN {X 0,Y 322.2,Z 403.221,A -85,B 0,C 180,E1 -15780.15,E2 -15780.15} C_VEL
LIN {X 0,Y 314.977,Z 386.234,A -85,B 0,C 180,E1 -15781.359,E2 -15781.359} C_VEL
LIN {X 0,Y 308.335,Z 372.237,A -85,B 0,C 180,E1 -15782.537,E2 -15782.537} C_VEL
LIN {X 0,Y 305.561,Z 361.543,A -85,B 0,C 180,E1 -15786.075,E2 -15786.075} C_VEL
LIN {X 0,Y 305.498,Z 361.072,A -85,B 0,C 180,E1 -15786.372,E2 -15786.372} C_VEL
LIN {X 0,Y 305.495,Z 361.035,A -85,B 0,C 180,E1 -15790.099,E2 -15790.099} C_VEL
LIN {X 0,Y 305.528,Z 361.035,A -85,B 0,C 180,E1 -15793.634,E2 -15793.634} C_VEL
LIN {X 0,Y 305.518,Z 361.047,A -85,B 0,C 180,E1 -15797.398,E2 -15797.398} C_VEL
LIN {X 0,Y 305.502,Z 361.013,A -85,B 0,C 180,E1 -15801.601,E2 -15801.601} C_VEL
LIN {X 0,Y 305.454,Z 361.053,A -85,B 0,C 180,E1 -15804.886,E2 -15804.886} C_VEL
LIN {X 0,Y 305.444,Z 361.042,A -85,B 0,C 180,E1 -15808.353,E2 -15808.353} C_VEL
LIN {X 0,Y 305.511,Z 360.996,A -85,B 0,C 180,E1 -15811.113,E2 -15811.113} C_VEL
LIN {X 0,Y 305.562,Z 361.032,A -85,B 0,C 180,E1 -15814.087,E2 -15814.087} C_VEL
LIN {X 0,Y 305.491,Z 361.04,A -85,B 0,C 180,E1 -15818.402,E2 -15818.402} C_VEL
LIN {X 0,Y 305.58,Z 361.044,A -85,B 0,C 180,E1 -15821.217,E2 -15821.217} C_VEL
LIN {X 0,Y 305.639,Z 361.021,A -85,B 0,C 180,E1 -15825.348,E2 -15825.348} C_VEL
LIN {X 0,Y 305.63,Z 361.023,A -85,B 0,C 180,E1 -15829.399,E2 -15829.399} C_VEL
LIN {X 0,Y 305.803,Z 361.01,A -85,B 0,C 180,E1 -15832.074,E2 -15832.074} C_VEL
LIN {X 0,Y 305.682,Z 361.028,A -85,B 0,C 180,E1 -15834.723,E2 -15834.723} C_VEL
LIN {X 0,Y 305.951,Z 360.993,A -85,B 0,C 180,E1 -15838.684,E2 -15838.684} C_VEL
LIN {X 0,Y 306.082,Z 360.982,A -85,B 0,C 180,E1 -15840,E2 -15840} C_VEL
LIN {X 0,Y 305.878,Z 360.991,A -85,B 0,C 180,E1 -15842.634,E2 -15842.634} C_VEL
LIN {X 0,Y 305.842,Z 361.012,A -85,B 0,C 180,E1 -15846.598,E2 -15846.598} C_VEL
LIN {X 0,Y 305.725,Z 361.005,A -85,B 0,C 180,E1 -15849.26,E2 -15849.26} C_VEL
LIN {X 0,Y 305.581,Z 361.039,A -85,B 0,C 180,E1 -15853.296,E2 -15853.296} C_VEL
LIN {X 0,Y 305.583,Z 361.023,A -85,B 0,C 180,E1 -15856.021,E2 -15856.021} C_VEL
LIN {X 0,Y 305.567,Z 361.04,A -85,B 0,C 180,E1 -15859.446,E2 -15859.446} C_VEL
LIN {X 0,Y 305.482,Z 361.054,A -85,B 0,C 180,E1 -15863.043,E2 -15863.043} C_VEL
LIN {X 0,Y 305.514,Z 361.033,A -85,B 0,C 180,E1 -15866.219,E2 -15866.219} C_VEL
LIN {X 0,Y 305.461,Z 361.001,A -85,B 0,C 180,E1 -15869.042,E2 -15869.042} C_VEL
LIN {X 0,Y 305.428,Z 361.05,A -85,B 0,C 180,E1 -15871.954,E2 -15871.954} C_VEL
LIN {X 0,Y 305.454,Z 361.053,A -85,B 0,C 180,E1 -15875.114,E2 -15875.114} C_VEL
LIN {X 0,Y 305.476,Z 361.017,A -85,B 0,C 180,E1 -15878.538,E2 -15878.538} C_VEL
LIN {X 0,Y 305.518,Z 361.047,A -85,B 0,C 180,E1 -15882.602,E2 -15882.602} C_VEL
LIN {X 0,Y 305.527,Z 361.035,A -85,B 0,C 180,E1 -15886.366,E2 -15886.366} C_VEL
LIN {X 0,Y 305.494,Z 361.035,A -85,B 0,C 180,E1 -15889.901,E2 -15889.901} C_VEL
LIN {X 0,Y 305.501,Z 361.125,A -85,B 0,C 180,E1 -15893.748,E2 -15893.748} C_VEL
LIN {X 0,Y 307.366,Z 368.424,A -85,B 0,C 180,E1 -15896.317,E2 -15896.317} C_VEL
LIN {X 0,Y 308.391,Z 372.376,A -85,B 0,C 180,E1 -15897.53,E2 -15897.53} C_VEL
LIN {X 0,Y 316.732,Z 390.064,A -85,B 0,C 180,E1 -15898.979,E2 -15898.979} C_VEL
LIN {X 0,Y 322.436,Z 403.869,A -85,B 0,C 180,E1 -15899.936,E2 -15899.936} C_VEL
LIN {X 0,Y 324.509,Z 415.767,A -85,B 0,C 180,E1 -15900.444,E2 -15900.444} C_VEL
LIN {X 0,Y 322.144,Z 494.247,A -85,B 0,C 180,E1 -15902.162,E2 -15902.162} C_VEL
LIN {X 0,Y 321.49,Z 512.526,A -85,B 0,C 180,E1 -15902.631,E2 -15902.631} C_VEL
LIN {X 0,Y 320.348,Z 526.897,A -85,B 0,C 180,E1 -15903.231,E2 -15903.231} C_VEL
LIN {X 0,Y 318.93,Z 540.132,A -85,B 0,C 180,E1 -15904.028,E2 -15904.028} C_VEL
LIN {X 0,Y 317.319,Z 553.543,A -85,B 0,C 180,E1 -15905.116,E2 -15905.116} C_VEL
LIN {X 0,Y 315.581,Z 565.632,A -85,B 0,C 180,E1 -15906.37,E2 -15906.37} C_VEL
LIN {X 0,Y 313.398,Z 577.827,A -85,B 0,C 180,E1 -15907.939,E2 -15907.939} C_VEL
LIN {X 0,Y 311.474,Z 587.899,A -85,B 0,C 180,E1 -15909.531,E2 -15909.531} C_VEL
LIN {X 0,Y 309.494,Z 597.909,A -85,B 0,C 180,E1 -15911.465,E2 -15911.465} C_VEL
LIN {X 0,Y 307.775,Z 606.698,A -85,B 0,C 180,E1 -15913.55,E2 -15913.55} C_VEL
LIN {X 0,Y 306.488,Z 614.164,A -85,B 0,C 180,E1 -15915.731,E2 -15915.731} C_VEL
LIN {X 0,Y 305.154,Z 620.556,A -85,B 0,C 180,E1 -15918.039,E2 -15918.039} C_VEL
LIN {X 0,Y 304.303,Z 626.224,A -85,B 0,C 180,E1 -15920.698,E2 -15920.698} C_VEL
LIN {X 0,Y 303.83,Z 630.336,A -85,B 0,C 180,E1 -15923.36,E2 -15923.36} C_VEL
LIN {X 0,Y 303.607,Z 633.015,A -85,B 0,C 180,E1 -15926.02,E2 -15926.02} C_VEL
LIN {X 0,Y 303.526,Z 634.338,A -85,B 0,C 180,E1 -15928.675,E2 -15928.675} C_VEL
LIN {X 0,Y 303.526,Z 634.33,A -85,B 0,C 180,E1 -15931.328,E2 -15931.328} C_VEL
LIN {X 0,Y 303.604,Z 633,A -85,B 0,C 180,E1 -15933.984,E2 -15933.984} C_VEL
LIN {X 0,Y 303.903,Z 631.429,A -85,B 0,C 180,E1 -15936.642,E2 -15936.642} C_VEL
LIN {X 0,Y 304.102,Z 630.078,A -85,B 0,C 180,E1 -15937.972,E2 -15937.972} C_VEL
LIN {X 0,Y 304.666,Z 627.201,A -85,B 0,C 180,E1 -15939.964,E2 -15939.964} C_VEL
LIN {X 0,Y 305.402,Z 623.289,A -85,B 0,C 180,E1 -15941.955,E2 -15941.955} C_VEL
LIN {X 0,Y 306.548,Z 618.221,A -85,B 0,C 180,E1 -15943.931,E2 -15943.931} C_VEL
LIN {X 0,Y 307.797,Z 611.908,A -85,B 0,C 180,E1 -15945.904,E2 -15945.904} C_VEL
LIN {X 0,Y 309.345,Z 604.128,A -85,B 0,C 180,E1 -15947.862,E2 -15947.862} C_VEL
LIN {X 0,Y 311.251,Z 594.585,A -85,B 0,C 180,E1 -15949.799,E2 -15949.799} C_VEL
LIN {X 0,Y 312.961,Z 584.936,A -85,B 0,C 180,E1 -15951.404,E2 -15951.404} C_VEL
LIN {X 0,Y 314.941,Z 573.162,A -85,B 0,C 180,E1 -15952.988,E2 -15952.988} C_VEL
LIN {X 0,Y 316.657,Z 560.575,A -85,B 0,C 180,E1 -15954.35,E2 -15954.35} C_VEL
